// All System Equipment
// Adjust GVL_EquipArrays.cEQUIP_COUNT_MAX to accommodate all of the equipment to monitor
IF GVL_EquipArrays.nSystemEquip_Count <> 0 THEN
	FOR nStatusArrayIndex := 1 TO GVL_EquipArrays.nSystemEquip_Count BY 1 DO
		IF nStatusArrayIndex <= GVL_EquipArrays.cEQUIP_COUNT_MAX THEN
			// Only process the equipment if is is not in an offline state, this allows for the separate PLC equipment to 
			IF GVL_EquipArrays.aSystemEquipStatusArray[nStatusArrayIndex].CrntState <> E_StateCntrl.stOffline THEN
				// Test for an active warning on a coveyor
				IF GVL_EquipArrays.aSystemEquipStatusArray[nStatusArrayIndex].StsHasWarnings THEN
					ConveyorHasWarn := 1;
				END_IF
				// Test for an active Equipment fault, more than just a conveyor fault, could include Remote/IO, Barcode reader, etc..
				IF GVL_EquipArrays.aSystemEquipStatusArray[nStatusArrayIndex].StsFaulted THEN
					ConveyorHasFault := 1;
				END_IF
				// Test for a sleeping state
				IF GVL_EquipArrays.aSystemEquipStatusArray[nStatusArrayIndex].CrntOperState = E_OperStateCntrl.sleeping THEN
					ConveyorIsSleeping := 1;
				END_IF
				// Test for the Auto state, again an equipment state test to include non-conveyor equipment
				IF GVL_EquipArrays.aSystemEquipStatusArray[nStatusArrayIndex].StsAuto THEN
					ConveyorInAuto := 1;
				END_IF
			END_IF
		END_IF
	END_FOR
END_IF

// Initialise the Stack Light, only changing values as required
//GVL_IO.LT_MainPanelStack_Blue := FALSE;
GVL_IO.LT_MainPanelStack_Green := FALSE;
GVL_IO.LT_MainPanelStack_Yellow := FALSE;
GVL_IO.LT_MainPanelStack_Red := FALSE;
GVL_IO.LT_10161_Red := FALSE;
GVL_IO.LT_3131_Red := FALSE;
GVL_IO.LT_8181_Red := FALSE;
GVL_IO.LT_10171_Yellow := FALSE;
GVL_IO.LT_3151_Yellow := FALSE;
GVL_IO.LT_8191_Yellow := FALSE;
GVL_IO.LT_10201_Green := FALSE;
GVL_IO.LT_3201_Green := FALSE;
GVL_IO.LT_8231_Green := FALSE;
	
IF ConveyorHasFault OR NOT SystemSafety.Safety_SystemEstopsOK THEN
	// Red light SOLID ON
	GVL_IO.LT_MainPanelStack_Red := TRUE;
	GVL_IO.LT_10161_Red := TRUE;
	GVL_IO.LT_3131_Red := TRUE;
	GVL_IO.LT_8181_Red := TRUE;
ELSE
	IF ConveyorHasWarn THEN
		// Orange Light SOLID ON
		GVL_IO.LT_MainPanelStack_Yellow := TRUE;
		GVL_IO.LT_10171_Yellow := TRUE;
		GVL_IO.LT_3151_Yellow := TRUE;
		GVL_IO.LT_8191_Yellow := TRUE;
	ELSE
		IF ConveyorInAuto THEN
			// Green Light SOLID ON
			GVL_IO.LT_MainPanelStack_Green := TRUE;
			GVL_IO.LT_10201_Green := TRUE;
			GVL_IO.LT_3201_Green := TRUE;
			GVL_IO.LT_8231_Green := TRUE;
		ELSE
			GVL_IO.LT_MainPanelStack_Green := SysShrtPulseTmr.Output;
			GVL_IO.LT_10201_Green :=  SysShrtPulseTmr.Output;
			GVL_IO.LT_3201_Green :=  SysShrtPulseTmr.Output;
			GVL_IO.LT_8231_Green :=  SysShrtPulseTmr.Output;
		END_IF
	END_IF
	IF GVL_IO.HornMainPanel THEN
		// Orange Light FLASHING ON
		GVL_IO.LT_MainPanelStack_Yellow := SysShrtPulseTmr.Output;
		GVL_IO.LT_10171_Yellow := SysShrtPulseTmr.Output;
		GVL_IO.LT_3151_Yellow := SysShrtPulseTmr.Output;
		GVL_IO.LT_8191_Yellow := SysShrtPulseTmr.Output;
	END_IF;
END_IF

END_PROGRAM

// ---- FunctionBlocks/Utils/FB_SystemCntrl.TcPOU
FUNCTION_BLOCK FB_SystemCntrl

(* System Interlock and Event Set up,
	Uses Interlocks.
	Doesn't use Start Conditions or the horn delay  
	Uses Events
	
	This exists to allow the Interlock/Event descriptions and setup to be managed through the HMI
	and be easily setup as system faults.
*)
VAR_IN_OUT
	{attribute 'OPC.UA.DA' := '1'}
	Sts_EquipState				: ST_EquipmentStatus;		// State Status
END_VAR
VAR_INPUT
	{attribute 'OPC.UA.DA' := '1'}
	In_o_EquipStatePB			: ST_StateCntrlPB;		// Hmi push buttons to change states
	In_p_EquipStatePB			: ST_StateCntrlPB;		// Other push buttons to change states
	{attribute 'OPC.UA.DA' := '1'}
	Cfg_EquipLabel				: STRING(20);		// Label of the equipment
	// Events
	In_SystemEvents				: UINT;		// Event that is specific to the instance of the solenoid/actuator
	{attribute 'OPC.UA.DA' := '0'}
	Cfg_EquipEvntsArry			: ARRAY [0..15] OF ST_CfgEvents;
	
	// Interlocks that can be Instance Specific
	In_SystemIntlks				: UINT;		// Interlock that is specific to the instance of the solenoid/actuator
	{attribute 'OPC.UA.DA' := '0'}
	Cfg_EquipIntlksArry		: ARRAY [0..15] OF ST_CfgEvents;		// Descriptions of the Interlock 
	
END_VAR
VAR_OUTPUT
	{attribute 'OPC.UA.DA' := '1'}
	Out_Auto					:	BOOL;	// Combine HMI and Other Start/Auto signals to issue a single START/AUTO command
	{attribute 'OPC.UA.DA' := '1'}
	Out_Stop					:	BOOL;	// Combine HMI and Other Stop signals to issue a single STOP command
	{attribute 'OPC.UA.DA' := '1'}
	Out_Reset					:	BOOL;	// Combine HMI and Other Reset signals to issue a single RESET command
	{attribute 'OPC.UA.DA' := '1'}
	Sts_All_Intlks_OK			: BOOL;		// Status bit to show that all interloks are good to Run 
	{attribute 'OPC.UA.DA' := '1'}
	Sts_FaultActive				: BOOL;	// Status Bit Showing that a fault is present (0= No Active Faults, 1= Fault Active)
	{attribute 'OPC.UA.DA' := '1'}
	Sts_WarnActive				: BOOL;	// Status Bit Showing that a warning is present (0= No Active Warnings, 1= Warning Active)
	{attribute 'OPC.UA.DA' := '1'}
	Sts_All_Evnts_OK			: BOOL;		// Status Bit Showing that ALL Events are OK to RUN (0= Event Present, 1= OK to Run)
	{attribute 'OPC.UA.DA' := '1'}
	Sts_IntlksArry				: ARRAY[0..15] OF ST_EventSts;		// Interlock status 0 to 15 Input
	{attribute 'OPC.UA.DA' := '1'}
	Sts_FaultsArry				: ARRAY[0..15] OF ST_EventSts;	// Status of each Fault Event State (0= OFF, 1=ON)
	{attribute 'OPC.UA.DA' := '1'}
	Sts_WarnsArry				: ARRAY[0..15] OF ST_EventSts;		// Status of each Warning Event State (0= OFF, 1=ON)
	{attribute 'OPC.UA.DA' := '0'}
	Sts_EvntsArry				: ARRAY[0..15] OF ST_EventSts; 	// Status of each Event State (0= OFF, 1=ON)
END_VAR
VAR
	{attribute 'OPC.UA.DA' := '0'}
	System_fbIntrlks				: FB_Intlks_Latch;
	System_IntlksArry				: ARRAY[0..15] OF BOOL;
	{attribute 'OPC.UA.DA' := '0'}
	System_EventManager				: FB_EventMngr;
	System_EventArry				: ARRAY[0..15] OF BOOL;
	System_LatchIgnore				: BOOL := FALSE;		// Put as a place holder for ease of future use
	System_LatchReset				: BOOL := FALSE;		//Put as a place holder for ease of future use
	System_IntlkBypassed			: ARRAY [0..15] OF BOOL;		//Put as a place holder for ease of future use
END_VAR

// Set Up inputs for interlocks that are specific for the configuration instance
System_IntlksArry[0] := In_SystemIntlks.0;
System_IntlksArry[1] := In_SystemIntlks.1; 
System_IntlksArry[2] := In_SystemIntlks.2;
System_IntlksArry[3] := In_SystemIntlks.3;
System_IntlksArry[4] := In_SystemIntlks.4;
System_IntlksArry[5] := In_SystemIntlks.5;
System_IntlksArry[6] := In_SystemIntlks.6;
System_IntlksArry[7] := In_SystemIntlks.7;
System_IntlksArry[8] := In_SystemIntlks.8;
System_IntlksArry[9] := In_SystemIntlks.9; 
System_IntlksArry[10] := In_SystemIntlks.10;
System_IntlksArry[11] := In_SystemIntlks.11;
System_IntlksArry[12] := In_SystemIntlks.12;
System_IntlksArry[13] := In_SystemIntlks.13;
System_IntlksArry[14] := In_SystemIntlks.14;
System_IntlksArry[15] := In_SystemIntlks.15;
	
// Call Interlock block
System_fbIntrlks(
	In_Intlks:= System_IntlksArry,
	CFG_IntlksArry:= Cfg_EquipIntlksArry, 
	HMI_LatchIgnore:= System_LatchIgnore, 
	HMI_LatchReset:= System_LatchReset, 
	All_Intlk_OK=> Sts_All_Intlks_OK, 
	STS_Intlks=> Sts_IntlksArry);
	
System_EventArry[0]:= In_SystemEvents.0;
System_EventArry[1]:= In_SystemEvents.1;
System_EventArry[2]:= In_SystemEvents.2;
System_EventArry[3]:= In_SystemEvents.3;
System_EventArry[4]:= In_SystemEvents.4;
System_EventArry[5]:= In_SystemEvents.5;
System_EventArry[6]:= In_SystemEvents.6;
System_EventArry[7]:= In_SystemEvents.7;
System_EventArry[8]:= In_SystemEvents.8;
System_EventArry[9]:= In_SystemEvents.9;
System_EventArry[10]:= In_SystemEvents.10;
System_EventArry[11]:= In_SystemEvents.11;
System_EventArry[12]:= In_SystemEvents.12;
System_EventArry[13]:= In_SystemEvents.13;
System_EventArry[14]:= In_SystemEvents.14;
System_EventArry[15]:= In_SystemEvents.15;

// Event Manager
System_EventManager(
	sEquipStateCntrlSts := Sts_EquipState.Sts_EquipmentState,
	In_EventsArry := System_EventArry ,  
	CFG_EvntsArry:= Cfg_EquipEvntsArry, 
	HMI_LatchReset:= In_o_EquipStatePB.ResetPB OR In_p_EquipStatePB.ResetPB,
	Out_FaultActive=> Sts_FaultActive, 
	Out_WarnActive=> Sts_WarnActive, 
	Sts_All_Evnts_OK=> Sts_All_Evnts_OK, 
	Sts_FaultsArry=> Sts_FaultsArry, 
	Sts_WarnsArry=> Sts_WarnsArry, 
	Sts_EvntsArry=> Sts_EvntsArry);

// Activate the Out_ variables
Out_Auto := In_o_EquipStatePB.AutoPB OR In_p_EquipStatePB.AutoPB;
Out_Stop := In_o_EquipStatePB.StopPB OR In_p_EquipStatePB.StopPB;
Out_Reset := In_o_EquipStatePB.ResetPB OR In_p_EquipStatePB.ResetPB;

// Populate the Sts Output Variables
Sts_EquipState.Sts_EquipmentState.CrntState := 1;
Sts_EquipState.Sts_All_Intlks_OK  := Sts_All_Intlks_OK;
Sts_EquipState.Sts_All_Evnts_OK  := Sts_All_Evnts_OK;
Sts_EquipState.Sts_FaultActive := Sts_FaultActive;
Sts_EquipState.Sts_WarnActive := Sts_WarnActive;

END_FUNCTION_BLOCK

// ---- FunctionBlocks/Utils/Events/FB_Intlks_Latch.TcPOU
FUNCTION_BLOCK FB_Intlks_Latch
(*
=====================================================================
	Copyright ©  Syscon Automation.  All Rights Reserved.
	Version 1 Release 1 2018
=====================================================================
 
	This FB monitors 16 interlock inputs
	Each "Good or OK" State for each Interlock Input is configurable (Default is 0=OK, 1=trip)
	Interlocks may be configured to latch which require a Reset Command to clear (latching can be disabled)
	Interlocks may be configured as Bypassable.
 --------------------------------------------------------------------
*)
 
VAR_INPUT
	In_Intlks:	ARRAY[0..15] OF BOOL;		// Interlocks 0 to 15 Input
	CFG_IntlksArry:	ARRAY[0..15] OF ST_CfgEvents;		// Configuration of Interlocks
	HMI_LatchIgnore:	BOOL;		// Input to ignore all latching requirements
	HMI_LatchReset:	BOOL;		// Input to reset latching interlocks
END_VAR
VAR_OUTPUT
	All_Intlk_OK: BOOL;		// Status Bit Showing that ALL Interlocks are OK to RUN (either interlock is OK or it has been bypassed (0= Interlock Enabled-Stop, 1= OK to Run)	
	STS_Intlks:	ARRAY[0..15] OF ST_EventSts;		// Status of each Interlock State (0= OFF, 1=ON)
	STS_LatchResetReq:	BOOL;		// Status bit to show that latch reset is req
	STS_BypassActive: BOOL;		// Status Bit Showing that a Bypass is Active (0= No Active Bypass, 1= A Bypass is Active) 
	
END_VAR
VAR
	Intlk_CrntStsArry:	ARRAY[0..15] OF BOOL;		// The Current state of the interlock after compared to OK state
	Intlks_LatchedArry:	ARRAY[0..15] OF BOOL;		//Currently Latched ON
	Intlks_Bypassed:	ARRAY[0..15] OF BOOL;		// Interlocks where Bypass is ON and Allowed
	STS_LatchResetReqArry:	ARRAY[0..15] OF BOOL; 		// Status to see if latch reset is required (0= OFF, 1=ON)
	Sts_Intlks_BypassNotAllowed:	ARRAY[0..15] OF BOOL;		// Status representing each Non Bypassable Interlock State (0= OFF, 1=ON)
	IntlkRaw_ON:	BOOL;		// Testing Bit to Show that an Interlock is Active Based on Current OK State (ignoring Latches and Bypassing)
	Intlk_ON:	BOOL;		// Testing Bit to Show that an Interlock is Active Based on Current OK State (After Latches and Bypassing)
	i: INT;		//index
END_VAR

// Run loop to check each input
FOR i := 0 TO 15 DO
	// Compare to OK State
	Intlk_CrntStsArry[i] := In_Intlks[i] XOR CFG_IntlksArry[i].OKState;
	
	//Look at Latching
	IF HMI_LatchIgnore THEN
		Intlks_LatchedArry[i] := Intlk_CrntStsArry[i];
	ELSE
		Intlks_LatchedArry[i] := Intlk_CrntStsArry[i] OR CFG_IntlksArry[i].LatchRequired; 			
	END_IF
	
	//Set Status based on Latching
	STS_Intlks[i].Status := (STS_Intlks[i].Status AND Intlks_LatchedArry[i]) OR Intlk_CrntStsArry[i];
	STS_LatchResetReqArry[i] := (STS_Intlks[i].Status AND Intlks_LatchedArry[i] AND CFG_IntlksArry[i].LatchRequired);
	
	//Look for Bypass State
	Intlks_Bypassed[i] := CFG_IntlksArry[i].ByPssAllwd AND CFG_IntlksArry[i].HMI_BypassPB; 
	Sts_Intlks_BypassNotAllowed[i] := NOT Intlks_Bypassed[i];  
	Sts_Intlks_BypassNotAllowed[i] := Sts_Intlks_BypassNotAllowed[i] AND STS_Intlks[i].Status;
	
	//Update Status based on bypass
	STS_Intlks[i].Status := STS_Intlks[i].Status AND (NOT Intlks_Bypassed[i]);
	STS_Intlks[i].Description := CFG_IntlksArry[i].Description;
	STS_Intlks[i].DeviceLabel := CFG_IntlksArry[i].DeviceLabel;
	IF STS_Intlks[i].Status AND STS_Intlks[i].Description <> '' THEN
		STS_Intlks[i].StatusTxt := 'TRUE';
	ELSE
		STS_Intlks[i].StatusTxt := 'FALSE';
	END_IF
END_FOR

IF HMI_LatchReset THEN
	FOR i := 0 TO 15 DO
		STS_Intlks[i].Status := FALSE;
		STS_LatchResetReqArry[i] := FALSE;
	END_FOR
END_IF

//Set Up test bit showing all active interlocks ignoring
IntlkRaw_ON := In_Intlks[0] OR In_Intlks[1] OR In_Intlks[2] OR In_Intlks[3] 
			OR In_Intlks[4]OR In_Intlks[5] OR In_Intlks[6] OR In_Intlks[7]
			OR In_Intlks[8] OR In_Intlks[9] OR In_Intlks[10] OR In_Intlks[11]
			OR In_Intlks[12] OR In_Intlks[13] OR In_Intlks[14] OR In_Intlks[15];
			
// Set up bit showing that All interlocks are good			
Intlk_ON := STS_Intlks[0].Status OR STS_Intlks[1].Status OR STS_Intlks[2].Status OR STS_Intlks[3].Status
			OR STS_Intlks[4].Status OR STS_Intlks[5].Status OR STS_Intlks[6].Status OR STS_Intlks[7].Status
			OR STS_Intlks[8].Status OR STS_Intlks[9].Status OR STS_Intlks[10].Status OR STS_Intlks[11].Status
			OR STS_Intlks[12].Status OR STS_Intlks[13].Status OR STS_Intlks[14].Status OR STS_Intlks[15].Status;
	
//Set Up test bit showing that a latch is required
STS_LatchResetReq := NOT HMI_LatchIgnore AND (STS_LatchResetReqArry[0] OR STS_LatchResetReqArry[1] OR STS_LatchResetReqArry[2] OR STS_LatchResetReqArry[3] 
			OR STS_LatchResetReqArry[4]OR STS_LatchResetReqArry[5] OR STS_LatchResetReqArry[6] OR STS_LatchResetReqArry[7]
			OR STS_LatchResetReqArry[8] OR STS_LatchResetReqArry[9] OR STS_LatchResetReqArry[10] OR STS_LatchResetReqArry[11]
			OR STS_LatchResetReqArry[12] OR STS_LatchResetReqArry[13] OR STS_LatchResetReqArry[14] OR STS_LatchResetReqArry[15]);
						
// Set up bit showing that a bypass is active			
STS_BypassActive := Intlks_Bypassed[0] OR Intlks_Bypassed[1] OR Intlks_Bypassed[2] OR Intlks_Bypassed[3]
			OR Intlks_Bypassed[4] OR Intlks_Bypassed[5] OR Intlks_Bypassed[6] OR Intlks_Bypassed[7]
			OR Intlks_Bypassed[8] OR Intlks_Bypassed[9] OR Intlks_Bypassed[10] OR Intlks_Bypassed[11]
			OR Intlks_Bypassed[12] OR Intlks_Bypassed[13] OR Intlks_Bypassed[14] OR Intlks_Bypassed[15];
			
// Set up bit showing that All interlocks are good			
All_Intlk_OK := NOT( STS_Intlks[0].Status OR STS_Intlks[1].Status OR STS_Intlks[2].Status OR STS_Intlks[3].Status
			OR STS_Intlks[4].Status OR STS_Intlks[5].Status OR STS_Intlks[6].Status OR STS_Intlks[7].Status
			OR STS_Intlks[8].Status OR STS_Intlks[9].Status OR STS_Intlks[10].Status OR STS_Intlks[11].Status
			OR STS_Intlks[12].Status OR STS_Intlks[13].Status OR STS_Intlks[14].Status OR STS_Intlks[15].Status);

END_FUNCTION_BLOCK

// ---- FunctionBlocks/Utils/Events/FB_EventMngr.TcPOU
FUNCTION_BLOCK FB_EventMngr
(*
=====================================================================
	Copyright ©  Syscon Automation.  All Rights Reserved.
	Version 1 Release 2 2020
=====================================================================
 
	This FB monitors 16 Event inputs
	Each "Good or OK" State for each Event Input is configurable (Default is 0=OK, 1=trip)
	Events may be configured to latch which require a Reset Command to clear (latching can be disabled)
	Events may be configured as Warnings or Alarms)

	Release Notes: 2 - Added Equipment state/control/status reference and Stop codes to record Faults/Warnings to report to the System
						The Equipment reference was added because just adding the stop register as an array cannot compile (3.1.4022.32)
 --------------------------------------------------------------------
*)
VAR_IN_OUT
	sEquipStateCntrlSts: ST_StateCntrlSts;		// Equipment State, Control and Status Object
END_VAR 
VAR_INPUT
	In_EventsArry:	ARRAY[0..15] OF BOOL;		// Events 0 to 15 Input	
	CFG_EvntsArry:	ARRAY[0..15] OF ST_CfgEvents;		// Event Configuration 
	HMI_LatchIgnore:	BOOL;		// Input to ignore all latching requirements
	HMI_LatchReset:	BOOL;		// Input to reset latching Event
	
END_VAR
VAR_OUTPUT	
	Out_FaultActive:	BOOL;	// Status Bit Showing that a fault is present (0= No Active Faults, 1= Fault Active)
	Out_WarnActive:	BOOL;	// Status Bit Showing that a warning is present (0= No Active Warnings, 1= Warning Active)
	Sts_All_Evnts_OK: BOOL;		// Status Bit Showing that ALL Events are OK to RUN (0= Event Present, 1= OK to Run)
	Sts_FaultsArry:	ARRAY[0..15] OF ST_EventSts;		// Status of each Fault Event State (0= OFF, 1=ON)
	Sts_WarnsArry:	ARRAY[0..15] OF ST_EventSts;		// Status of each Warning Event State (0= OFF, 1=ON)
	Sts_EvntsArry:	ARRAY[0..15] OF ST_EventSts;		// Status of each Event State (0= OFF, 1=ON)
	Sts_LatchResetReq:	BOOL;		// Status bit to show that latch reset is req
	Sts_StopCode: UINT;				// Highest Priority Stop Code (Lowest Bit Weight)
	
END_VAR
VAR
	Evnt_CrntStsArry:	ARRAY[0..15] OF BOOL;		// The Current state of the Event after compared to OK state
	Evnts_LatchedArry:	ARRAY[0..15] OF BOOL;		//Currently Latched ON
	STS_LatchResetReqArry:	ARRAY[0..15] OF BOOL; 		// Status to see if latch reset is required (0= OFF, 1=ON)

	Evnt_ON:	BOOL;		// Testing Bit to Show that an Event is Active Based on Current OK State (ignoring Latches and Bypassing)
	i: INT;		//index
	fb_ManageStopCodes	:	FB_ManageCodes;			// Function Block with Methods to manage codes

	Evnt_Delay:		ARRAY[0..15] OF Tc2_Standard.TON;	// Set of timers to Delay configured events
	DelayTest:	DWORD;
END_VAR

// Clear the Sts_StopCode each pass
Sts_StopCode := 0;

// Run loop to check each input
FOR i := 0 TO 15 DO

	// Only "Online" items can be faulted
	IF sEquipStateCntrlSts.CrntState <> E_StateCntrl.stOffline THEN
		// Test for a value in the EventDelay
		DelayTest := TIME_TO_DWORD(CFG_EvntsArry[i].EventDelay); 
		IF ( DelayTest > 0) THEN
			Evnt_Delay[i].PT := CFG_EvntsArry[i].EventDelay;
			Evnt_Delay[i].IN := In_EventsArry[i] XOR CFG_EvntsArry[i].OKState;
			Evnt_Delay[i]();
			Evnt_CrntStsArry[i] := Evnt_Delay[i].Q;
		ELSE
			// Compare to OK State, if they match, the CrntStsArry is = 0
			//  1 XOR 1 = 0, 1 XOR 0 = 1, 0 XOR 1 = 1, 0 XOR 0 = 0 
			Evnt_CrntStsArry[i] := In_EventsArry[i] XOR CFG_EvntsArry[i].OKState;
		END_IF
	ELSE
		Evnt_CrntStsArry[i] := FALSE;
	END_IF
	
	//Look at Latching
	// HMI_LatchIgnore latches ALL Events, over-riding the Latch setup per event
	IF HMI_LatchIgnore THEN
		Evnts_LatchedArry[i] := Evnt_CrntStsArry[i];
	ELSE
		Evnts_LatchedArry[i] := Evnt_CrntStsArry[i] OR CFG_EvntsArry[i].LatchRequired; 			
	END_IF
	
	//Set Status based on Latching
	Sts_EvntsArry[i].Status := (Sts_EvntsArry[i].Status AND Evnts_LatchedArry[i]) OR Evnt_CrntStsArry[i];
	Sts_EvntsArry[i].Description := CFG_EvntsArry[i].Description;
	Sts_EvntsArry[i].DeviceLabel := CFG_EvntsArry[i].DeviceLabel;	
	STS_LatchResetReqArry[i] := (Sts_EvntsArry[i].Status AND Evnts_LatchedArry[i] AND CFG_EvntsArry[i].LatchRequired);
	IF Sts_EvntsArry[i].Status AND Sts_EvntsArry[i].Description <> '' THEN
		Sts_EvntsArry[i].StatusTxt := 'TRUE';
	ELSE
		Sts_EvntsArry[i].StatusTxt := 'FALSE';
	END_IF
	
	//Seperate into Alarms and Faults 
	Sts_FaultsArry[i].Status := Sts_EvntsArry[i].Status AND CFG_EvntsArry[i].FaultWarn;
	Sts_FaultsArry[i].Description := Sts_EvntsArry[i].Description;
	Sts_FaultsArry[i].DeviceLabel := Sts_EvntsArry[i].DeviceLabel;
	IF Sts_FaultsArry[i].Status AND Sts_FaultsArry[i].Description <> '' THEN
		Sts_FaultsArry[i].StatusTxt := 'TRUE';
	ELSE
		Sts_FaultsArry[i].StatusTxt := 'FALSE';
	END_IF
	
	Sts_WarnsArry[i].Status := Sts_EvntsArry[i].Status AND (NOT CFG_EvntsArry[i].FaultWarn);
	Sts_WarnsArry[i].Description := Sts_EvntsArry[i].Description;
	Sts_WarnsArry[i].DeviceLabel := Sts_EvntsArry[i].DeviceLabel;	
	IF Sts_WarnsArry[i].Status AND Sts_WarnsArry[i].Description <> '' THEN
		Sts_WarnsArry[i].StatusTxt := 'TRUE';
	ELSE
		Sts_WarnsArry[i].StatusTxt := 'FALSE';
	END_IF

	// Instanciate the fb_ManageStopCodes Function Block
	fb_ManageStopCodes(aCodeRegister := sEquipStateCntrlSts.stsStopRegister);

	// Check for a configured stop code
	IF CFG_EvntsArry[i].StopCode <> 0  THEN
		// Set the Stop Register for the configured stop code
		IF Sts_EvntsArry[i].Status THEN
			// Lowest Stop Code is highest Priority
			IF (Sts_StopCode > CFG_EvntsArry[i].StopCode) THEN
				Sts_StopCode := CFG_EvntsArry[i].StopCode;
			END_IF
			fb_ManageStopCodes.Set(nCodeToSet := CFG_EvntsArry[i].StopCode);
		ELSE
			// Clear the Stop Register for non-latching Events, when the HMI_LatchIgnore is NOT set
			IF NOT (CFG_EvntsArry[i].LatchRequired) AND NOT HMI_LatchIgnore THEN
				fb_ManageStopCodes.Clear(nCodeToClear := CFG_EvntsArry[i].StopCode);
			END_IF
		END_IF
	END_IF
	
END_FOR

IF HMI_LatchReset OR (sEquipStateCntrlSts.CrntState = E_StateCntrl.stOffline) THEN
	FOR i := 0 TO 15 DO
		Sts_EvntsArry[i].Status := FALSE;
		STS_LatchResetReqArry[i] := FALSE;
	END_FOR
	// When the Reset is issued, clear the entire stop register
	fb_ManageStopCodes.ClearRegister();
END_IF

//Set Up test bit showing all active Event ignoring bypasses and latching
Evnt_ON := In_EventsArry[0] OR In_EventsArry[1] OR In_EventsArry[2] OR In_EventsArry[3] 
			OR In_EventsArry[4]OR In_EventsArry[5] OR In_EventsArry[6] OR In_EventsArry[7]
			OR In_EventsArry[8] OR In_EventsArry[9] OR In_EventsArry[10] OR In_EventsArry[11]
			OR In_EventsArry[12] OR In_EventsArry[13] OR In_EventsArry[14] OR In_EventsArry[15];
			
//Set Up test bit showing that a latch is required
STS_LatchResetReq := NOT HMI_LatchIgnore AND (STS_LatchResetReqArry[0] OR STS_LatchResetReqArry[1] OR STS_LatchResetReqArry[2] OR STS_LatchResetReqArry[3] 
			OR STS_LatchResetReqArry[4]OR STS_LatchResetReqArry[5] OR STS_LatchResetReqArry[6] OR STS_LatchResetReqArry[7]
			OR STS_LatchResetReqArry[8] OR STS_LatchResetReqArry[9] OR STS_LatchResetReqArry[10] OR STS_LatchResetReqArry[11]
			OR STS_LatchResetReqArry[12] OR STS_LatchResetReqArry[13] OR STS_LatchResetReqArry[14] OR STS_LatchResetReqArry[15]);
						
// Set up bit showing that All Event are good			
STS_All_Evnts_OK := NOT( Sts_EvntsArry[0].Status OR Sts_EvntsArry[1].Status OR Sts_EvntsArry[2].Status OR Sts_EvntsArry[3].Status
			OR Sts_EvntsArry[4].Status OR Sts_EvntsArry[5].Status OR Sts_EvntsArry[6].Status OR Sts_EvntsArry[7].Status
			OR Sts_EvntsArry[8].Status OR Sts_EvntsArry[9].Status OR Sts_EvntsArry[10].Status OR Sts_EvntsArry[11].Status
			OR Sts_EvntsArry[12].Status OR Sts_EvntsArry[13].Status OR Sts_EvntsArry[14].Status OR Sts_EvntsArry[15].Status);

// Set up bit showing A Fault is Active			
Out_FaultActive := Sts_FaultsArry[0].Status OR Sts_FaultsArry[1].Status OR Sts_FaultsArry[2].Status OR Sts_FaultsArry[3].Status
			OR Sts_FaultsArry[4].Status OR Sts_FaultsArry[5].Status OR Sts_FaultsArry[6].Status OR Sts_FaultsArry[7].Status
			OR Sts_FaultsArry[8].Status OR Sts_FaultsArry[9].Status OR Sts_FaultsArry[10].Status OR Sts_FaultsArry[11].Status
			OR Sts_FaultsArry[12].Status OR Sts_FaultsArry[13].Status OR Sts_FaultsArry[14].Status OR Sts_FaultsArry[15].Status;
			
// Set up bit showing A Warning is Active			
Out_WarnActive :=  Sts_WarnsArry[0].Status OR Sts_WarnsArry[1].Status OR Sts_WarnsArry[2].Status OR Sts_WarnsArry[3].Status
			OR Sts_WarnsArry[4].Status OR Sts_WarnsArry[5].Status OR Sts_WarnsArry[6].Status OR Sts_WarnsArry[7].Status
			OR Sts_WarnsArry[8].Status OR Sts_WarnsArry[9].Status OR Sts_WarnsArry[10].Status OR Sts_WarnsArry[11].Status
			OR Sts_WarnsArry[12].Status OR Sts_WarnsArry[13].Status OR Sts_WarnsArry[14].Status OR Sts_WarnsArry[15].Status;

END_FUNCTION_BLOCK

// ---- FunctionBlocks/StateControl/FB_ManageCodes.TcPOU
FUNCTION_BLOCK FB_ManageCodes
VAR_IN_OUT
	aCodeRegister: ARRAY[*] OF UDINT;	// Variable array for Different sizes of Code Registers
END_VAR
VAR_INPUT
END_VAR
VAR_OUTPUT
END_VAR
VAR
	nBitIndex : UINT;						// Bit within the Word
	nArrayIndex : UINT;						// Word within the array
	nArrayTempIndex : UINT;					// Array Index for processing array
	nArrayCount : UINT;						// Number of words in the Array
	nUpdateValue : UDINT;					// Value of the Word to OR/XOR with the 
	nCheckValue : UDINT;					// Value of the Word to check with
	nBitCheck : UDINT;						// Word to use to check if a bit is set
	nLowerBitCheck : UDINT;					// Word to use to check if a lower weighted bit is set
END_VAR

VAR CONSTANT
	nBITCOUNT: UINT := 32;	// Number of Bits in each Array Element
	nBYTECOUNT : UINT := 4;	// Number of Bytes in each array element
END_VAR

// Get the array count
nArrayCount := (TO_UINT(SIZEOF(aCodeRegister)))/nBYTECOUNT;

METHOD PUBLIC Check : BOOL
VAR_INPUT
	nCodeToCheck : UINT;				// Code to Check For
END_VAR
VAR_OUTPUT
	bCodeSet : BOOL;					// Indicates that the Code is Set
	bHigherPriorityCode : BOOL;			// Indicates that a Higher Priority Code is Set
END_VAR
// Disable the warning regarding invalid Reference from a method for IO_OUT variables
{warning disable C0371}
// Test for a Valid reference
//IF __ISVALIDREF(aCodeRegister) THEN
	// Test to see if a bit is set
	nArrayIndex := 0;
	nBitIndex := 0;
	// Test for a valid value to test, > 0, < maximum number of available bits
	IF (nCodeToCheck <> 0) THEN
		IF nCodeToCheck <= (nArrayCount * nBITCOUNT) THEN
			// Use integer division to obtain the array index
			// Subtract 1 to put items in the range of 0-31 bits to use EXPT function to set individual bits (2^bit weight)
			nArrayIndex := (nCodeToCheck - 1) / nBITCOUNT;
			// Use modulo division to get the remainder that indicates the bit weight 
			nBitIndex := (nCodeToCheck - 1) MOD nBITCOUNT;
			// Calculate the value (2^nBitIndex)
			nCheckValue := TO_UDINT(EXPT(2,nBitIndex));
			// Bitwise AND the result with the target.
			// The AND clears all other bits in the word
			nBitCheck := aCodeRegister[nArrayIndex] AND nCheckValue;
			// The only bit that should survive the AND is the one we are checking for
			bCodeSet := (nBitCheck <> 0); 
		END_IF
	ELSE
		// Clear the Stop Code check when there is no request
		bCodeSet := 0;
	END_IF
	
	// Only test for a higher priority stop code if the tested stop code exists
	IF bCodeSet = 1 THEN
		// Test to see if a lower weighted bit is set
		nArrayIndex := 0;
		nBitIndex := 0;
		// Test for a valid value to test, > 0, < maximum number of available bits
		IF (nCodeToCheck <> 0) THEN
			IF nCodeToCheck <= (nArrayCount * nBITCOUNT) THEN
				// Use integer division to obtain the array index
				// Subtract 1 to put items in the range of 0-31 bits to use EXPT function to set individual bits (2^bit weight)
				nArrayIndex := (nCodeToCheck - 1) / nBITCOUNT;
				// Use modulo division to get the remainder that indicates the bit weight 
				nBitIndex := (nCodeToCheck - 1) MOD nBITCOUNT;
				// Calculate the value (2^nBitIndex)
				nCheckValue := TO_UDINT(EXPT(2,nBitIndex));
				// Subtract 1 from the bit we are checking, this flips all the less significant bits
				// E.g. 4 (0100b) - 1 (0001b) = 3 (0011b)
				// E.g. 21 (10101b) - 1 (00001b) = 20 (10100b)
				// E.g. 24 (11000b) - 1 (00001b) = 23 (10111b)
				nCheckValue := nCheckValue - 1; 
				// The AND masks out all bits above the specified weight, including the one we are testing for
				//  leaving only bits with a lower bit weight
				nLowerBitCheck := aCodeRegister[nArrayIndex] AND nCheckValue;
				// Test the calculated value for a lower bit
				bHigherPriorityCode := (nLowerBitCheck <> 0); 
				// Test to see if we are in the lowest array
				nArrayTempIndex := 0;
				IF nArrayIndex <> 0 THEN
					WHILE nArrayTempIndex < nArrayIndex  DO
						IF aCodeRegister[nArrayTempIndex] <> 0 THEN
							bHigherPriorityCode := 1;
						END_IF
						nArrayTempIndex := nArrayTempIndex + 1;
					END_WHILE
				END_IF
			END_IF
		END_IF
	ELSE
		// Reset the higher priority detected if the Tested Stop Code is not set
		bHigherPriorityCode := 0;
	END_IF
//END_IF
// Restore the warning regarding invalid Reference from a method for IO_OUT variables
{warning restore C0371}
END_METHOD

METHOD PUBLIC Clear
VAR_INPUT
	nCodeToClear : UINT;					// Stop Code to Activate
END_VAR
// Disable the warning regarding invalid Reference from a method for IO_OUT variables
{warning disable C0371}
// Test for a Valid reference
//IF __ISVALIDREF(aCodeRegister) THEN
	// Clear an individual bit
	// Initialize the index values
	nArrayIndex := 0;
	nBitIndex := 0;
	// Test for a valid value to test, > 0, < maximum number of available bits
	IF (nCodeToClear <> 0) THEN
		IF nCodeToClear <= (nArrayCount * nBITCOUNT) THEN
			// Use integer division to obtain the array index
			// Subtract 1 to put items in the range of 0-31 bits to use EXPT function to set individual bits (2^bit weight)
			nArrayIndex := (nCodeToClear - 1) / nBITCOUNT;
			// Use modulo division to get the remainder that indicates the bit weight 
			nBitIndex := (nCodeToClear - 1) MOD nBITCOUNT;
			// Calculate the value (2^nStopCode)
			nUpdateValue := TO_UDINT(EXPT(2,nBitIndex));
			// Bitwise OR the result with the target.
			// The OR leaves all other bits in the word set, even the one to be set if it already is
			// In this instance, it ensures that the following XOR clears the bit
			// 0 XOR 0 = 0, 1 XOR 0 = 0, 1 XOR 1 = 0
			aCodeRegister[nArrayIndex] := aCodeRegister[nArrayIndex] OR nUpdateValue;
			aCodeRegister[nArrayIndex] := aCodeRegister[nArrayIndex] XOR nUpdateValue; 
		END_IF
	END_IF
//END_IF
// Restore the warning regarding invalid Reference from a method for IO_OUT variables
{warning restore C0371}
END_METHOD

METHOD PUBLIC ClearRegister
VAR_INPUT
END_VAR
// Disable the warning regarding invalid Reference from a method for IO_OUT variables
{warning disable C0371}
// Test for a Valid reference
//IF __ISVALIDREF(aCodeRegister) THEN
	// aCodeRegister is a Zero based array
	// The SIZEOF will return the 1 based number of elements
	// Decrement this by 1 (one) to process the array
	FOR nArrayIndex := 0 TO (nArrayCount - 1) BY 1 DO
		// Clear each register
		aCodeRegister[nArrayIndex] := 0;
	END_FOR
//END_IF
// Restore the warning regarding invalid Reference from a method for IO_OUT variables
{warning restore C0371}
END_METHOD

METHOD PUBLIC Set
VAR_INPUT
	nCodeToSet	:	UINT;
END_VAR
// Disable the warning regarding invalid Reference from a method for IO_OUT variables
{warning disable C0371}
// Test for a Valid reference
//IF __ISVALIDREF(aCodeRegister) THEN
	// Set an individual bit
	// Initialize the index values
	nArrayIndex := 0;
	nBitIndex := 0;
	// Test for a valid value to test, > 0, < maximum number of available bits
	IF (nCodeToSet <> 0) THEN
		IF nCodeToSet <= (nArrayCount * nBITCOUNT) THEN
			// Use integer division to obtain the array index
			// Subtract 1 to put items in the range of 0-31 bits to use EXPT function to set individual bits (2^bit weight)
			nArrayIndex := (nCodeToSet - 1) / nBITCOUNT;
			// Use modulo division to get the remainder that indicates the bit weight 
			nBitIndex := (nCodeToSet - 1) MOD nBITCOUNT;
			// Calculate the value (2^nStopCode)
			nUpdateValue := TO_UDINT(EXPT(2,nBitIndex));
			// Bitwise OR the result with the target.
			// The OR leaves all other bits in the word set, even the one to be set if it already is
			aCodeRegister[nArrayIndex] := aCodeRegister[nArrayIndex] OR nUpdateValue;
		END_IF
	END_IF
//END_IF
// Restore the warning regarding invalid Reference from a method for IO_OUT variables
{warning restore C0371}
END_METHOD

END_FUNCTION_BLOCK

// ---- FunctionBlocks/Utils/FB_Flasher.TcPOU
(*
Function Block to vreate a flashing output.
If In_Trig goes TRUE the output will begin to blink On and OFF until In_Trig goes FALSE.
On duration is set by Cfg_OnTime
Off duration is set by Cfg_OffTime
*)
FUNCTION_BLOCK FB_Flasher
VAR_INPUT
	In_Trig:	BOOL;		// Input Trigger (1= Flsh output based on configured time intrevals)
	Cfg_OnTime:	TIME;		// Output On Time
	Cfg_OffTime:	TIME;	// Output Off Time
END_VAR
VAR_OUTPUT
	Output:	BOOL;		// Flashing Output
END_VAR
VAR
	StartTrig: R_TRIG;		// Rising Trigger
	OnTmrActive: BOOL;		// ON Timer active
	OnTmr: TON;				// ON Timer
	OffTmrActive: BOOL;		// OFF Timer active
	OffTmr: TON;			// OFF Timer
	StopTrig: F_TRIG;		// Falling Trigger 
END_VAR

// Start on Rise
StartTrig(CLK:= In_Trig);

IF StartTrig.Q THEN
	OnTmrActive := TRUE;
END_IF

// On timer
OnTmr(IN:= OnTmrActive, PT:= Cfg_OnTime);
IF OnTmr.Q THEN
	OnTmrActive := FALSE;
	OffTmrActive := TRUE;
END_IF

// Off Timer 
OffTmr(IN:= OffTmrActive, PT:= Cfg_OffTime);
IF OffTmr.Q THEN
	OnTmrActive := TRUE;
	OffTmrActive := FALSE;
END_IF

// Stop Trigger
StopTrig(CLK:= In_Trig);

IF StopTrig.Q THEN
	OnTmrActive := FALSE;
	OffTmrActive := FALSE;
END_IF

// Set Output
Output := OnTmrActive AND In_Trig;

END_FUNCTION_BLOCK

// ---- FunctionBlocks/Utils/FB_AlrtStrtDelay.TcPOU
(*
Function block to sound an Alert or Horn while delaying the start up of a piece of equipment
Can be controlled by a start and stop pulse In_StrtPulse/In_StpPulse Or by a holding the run variable In_Run TRUE.
The delay times are configured by CFG_AlertTime and CFG_WaitTime
The delay can be bypassed by In_BypssDelay.
If the run signal is True or the Start Pulse is triggered the Alert is sounded for the Alert time.
After Alert time is elapsed the alert is set to False and the wait time is then started
at the completion of the wait time the output is set to TRUE and the Out_Pulse is held true for one scan
If the In_BypssDelay input is true then the output is set to true imediately with the run signal or start pulse.
The alert can be fired manually (without affecting the delays) at anytime using the In_ManTstTrig input.
*)
FUNCTION_BLOCK FB_AlrtStrtDelay
VAR_INPUT
	In_Run:	BOOL;				// Run signal that has to be held on to operate delay
	In_StrtPulse :	BOOL;		// Pulse or Triger to Start Delay
	In_StpPulse :	BOOL;		// Pulse or Triger to Stop Delay
	CFG_AlertTime:	TIME;		// Time (or duration) for the alert or Horn to sound
	CFG_WaitTime:	TIME;		// Time to delay after alert or horn has sounded
	CFG_PulseTime:	TIME;		// Time to pulse the output signal
	In_ManTstTrig:	BOOL;		// Manual bit to alert or sound horn for the time/duration 
	In_BypssDelay:	BOOL;		// Input to disable and bypass alert or horn delay
END_VAR
VAR_OUTPUT
	Out:	BOOL;		// Output that is delayed by the horn timers.  Latched On while Run is True Or if RUN is FALSE then until Stop Pulse.
	Out_Pulse:	BOOL;		// Output that is delayed by the horn timers.  Pulsed for one scan
	Out_Timed:	BOOL;		// Output that is delayed by the horn timers.  Pulsed for configurable amount of time
	Out_Alert:	BOOL;		// Output for the ALert or Horn
	Sts_DelayActive:	BOOL; // Status output to show when output is actively being delayed
END_VAR
VAR
	AlertRequired: BOOL := FALSE;
	WaitRequired: BOOL := FALSE;
	AlertTon: TON;
	WaitActive: BOOL := FALSE;
	WaitTon: TON;
	DelayCompleted: BOOL := FALSE;
	DelayComplete: BOOL := FALSE;
	StartTrig: R_TRIG;
	ManTrig: R_TRIG;
	StopTrig: F_TRIG;
	OutTrig: R_TRIG;
	OutTrigTOF: TOF; // Pulse the Start Trigger for a set period of time
END_VAR

// Start Alert or Horn
StartTrig(CLK:= In_Run OR In_StrtPulse AND NOT In_BypssDelay);
IF StartTrig.Q THEN
	AlertRequired := TRUE;
	WaitRequired :=TRUE;
	Sts_DelayActive := TRUE;
END_IF

ManTrig(CLK:= In_ManTstTrig);
IF ManTrig.Q THEN
	AlertRequired := TRUE;
	WaitRequired :=FALSE;
END_IF

// Sound horn for timer
AlertTon(IN:= AlertRequired , PT:=CFG_AlertTime);

IF AlertTon.Q THEN
	AlertRequired:= FALSE;
	IF WaitRequired THEN
		WaitActive:= TRUE;
		DelayComplete := FALSE;	
	ELSE
		WaitActive := FALSE;
		WaitRequired := FALSE;
		Sts_DelayActive := FALSE;
		DelayComplete := TRUE;	
	END_IF	
END_IF

WaitTon(IN:=WaitActive, PT:=CFG_WaitTime);
IF WaitTon.Q THEN
	WaitActive := FALSE;
	WaitRequired := FALSE;
	Sts_DelayActive := FALSE;
	DelayComplete := TRUE;
END_IF

// Reset on stop
StopTrig(CLK:= In_Run OR In_StpPulse);
IF StopTrig.Q THEN
	AlertRequired:= FALSE;
	WaitRequired := FALSE;
	WaitActive := FALSE;
	Sts_DelayActive := FALSE;
	DelayComplete := FALSE;
END_IF
		
//Set Output
Out_Alert := AlertRequired;
Out := DelayComplete OR (In_BypssDelay AND In_Run);
OutTrig(CLK:= OUT, Q=> Out_Pulse);

// Timed Output
OutTrigTOF(IN := OutTrig.Q, PT := CFG_PulseTime);
Out_Timed := OutTrigTOF.Q;

END_FUNCTION_BLOCK

// ---- POUs/BarCodeReaders.TcPOU
PROGRAM BarCodeReaders
VAR
	BCR_S2140_01: CognexDataMan260;		// P2140 Divert 
	BCR_S2141_01: CognexDataMan260;		// P2141 Location Update
	BCR_S2150_01: CognexDataMan260;		// P2150 Sorter	
	BCR_S3080_01: CognexDataMan260;		// P3080 Location Update

//----------------------------------------BCR_S2140_01--------------------------------------------------------------		
	P2140_Arrival_Item 			: ST_Item;		// Output Item (Bar code read) To Sort PLC
	P2140_LastArrival_Item		: ST_Item;		// Last Output Item (Bar code read) To Sort PLC
	ReadID_P2140_Old		: UDINT;

	fb_SorterArrivalBuffer_P2140			: FB_ItemBuffer;	// Function to Process the SorterArrivalBuffer
	
	sBcr2140Log			: STRING;
	tpBcr2140Trig					: TP;	// Pulse timer for BCR Reader

	rSorter2140PE					: R_TRIG; 	// Capture the Rising edge of the Sorter BCR PE
	fSorter2140PE					: F_TRIG; 	// Capture the Falling edge of the Sorter BCR PE
	r_BCR2140TriggerON			: R_TRIG;
	f_BCR2140TriggerON			: F_TRIG;
	
//----------------------------------------BCR_S2150_01--------------------------------------------------------------
	P2150_Arrival_Item 			: ST_Item;		// Output Item (Bar code read) To Sort PLC
	P2150_LastArrival_Item		: ST_Item;		// Last Output Item (Bar code read) To Sort PLC
	ReadID_P2150_Old		: UDINT;

	fb_SorterArrivalBuffer_P2150			: FB_ItemBuffer;	// Function to Process the SorterArrivalBuffer

	sBcr2150Log			: STRING;
	tpBcr2150Trig					: TP;	// Pulse timer for BCR Reader

	rSorter2150PE					: R_TRIG; 	// Capture the Rising edge of the Sorter BCR PE
	fSorter2150PE					: F_TRIG; 	// Capture the Falling edge of the Sorter BCR PE
	r_BCR2150TriggerON			: R_TRIG;
	f_BCR2150TriggerON			: F_TRIG;

END_VAR

(*
	When multiple origination requests are possible, create multiple arrival buffers, one per origination request
	Along with all of the required structures 
	These additional buffers are mapped as I/O between this routine and the corresponding ProcessBuffers program instance
*)
//----------------------------------------BCR_S2140_01--------------------------------------------------------------
// Create instances of Buffer Processing Functions to initialize the buffers and data
fb_SorterArrivalBuffer_P2140.Master := TRUE;

// Setup Logging
fb_SorterArrivalBuffer_P2140.LogEntries := .nItemBufferLogEnable.ARRIVALS OR .nItemBufferLogEnableP2140.ARRIVALS;

// Setup Buffer Name for Logging
fb_SorterArrivalBuffer_P2140.Name := 'P2140 SYS ARRIVAL';

fb_SorterArrivalBuffer_P2140(st_BufferData := st_SorterArrivalBuffer_P2140
					, st_BufferFdbkIn := st_ArrivalFdbkIn_P2140
					, st_BufferFdbkOut => st_ArrivalFdbkOut_P2140);

IF GVL_IO.INIT THEN
	fb_SorterArrivalBuffer_P2140.Clear();
END_IF
//----------------------------------------BCR_S2150_01--------------------------------------------------------------
// Create instances of Buffer Processing Functions to initialize the buffers and data
fb_SorterArrivalBuffer_P2150.Master := TRUE;

// Setup Logging
fb_SorterArrivalBuffer_P2150.LogEntries := .nItemBufferLogEnable.ARRIVALS OR .nItemBufferLogEnableP2150.ARRIVALS;

// Setup Buffer Name for Logging
fb_SorterArrivalBuffer_P2150.Name := 'P2150 SYS ARRIVAL';

fb_SorterArrivalBuffer_P2150(st_BufferData := st_SorterArrivalBuffer_P2150
					, st_BufferFdbkIn := st_ArrivalFdbkIn_P2150
					, st_BufferFdbkOut => st_ArrivalFdbkOut_P2150);

IF GVL_IO.INIT THEN
	fb_SorterArrivalBuffer_P2150.Clear();
END_IF


// Reset All Metrics when requested
IF MAIN.In_ResetAllMetrics THEN
	BCR_S2140_01.In_ResetCounts := MAIN.In_ResetAllMetrics;
	BCR_S2141_01.In_ResetCounts := MAIN.In_ResetAllMetrics;
	BCR_S2150_01.In_ResetCounts := MAIN.In_ResetAllMetrics;
	BCR_S3080_01.In_ResetCounts := MAIN.In_ResetAllMetrics;

END_IF
//----------------------------------------BCR_S2140_01--------------------------------------------------------------
//Divert
// Set up Bar Code Readers
BCR_S2140_01.LogEntries := .nBarcodeLogEnable.BCR_S2140_01_LOG;
BCR_S2140_01(
	In_ReadTrig:= PhotoEyes.PE_10081.Out_OnFltrd, 
	In_ResetCounts:= , 
	In_TriggerOnTime := T#20MS ,
	In_EquipID := '00064',
	Out_NewReadTrig=> , 
	Out_ReadString=> , 
	Out_ReadStatus=> ,
	Out_ResultID=>, 
	MisreadCount=> , 
	GoodreadCount=> );
//Logging
BCR_S2140_01.LogEntries := .nBarcodeLogEnable.BCR_S2140_01_LOG;
tpBcr2140Trig(
	IN := PhotoEyes.PE_10081.Out,
				PT := T#10MS,
				Q =>);
// Capture rising and falling edge Triggers of the Sorter BCR Trigger PE
rSorter2140PE(CLK:= PhotoEyes.PE_10081.Out, Q =>);
fSorter2140PE(CLK:= PhotoEyes.PE_10081.Out, Q =>);

// Log the rising/falling edge of the Trigger
IF rSorter2140PE.Q OR fSorter2140PE.Q THEN
	IF nBarcodeLogEnable.TRIGGER_PE THEN
		// Write to the Error List
		ADSLOGSTR( msgCtrlMask := ADSLOG_MSGTYPE_HINT OR ADSLOG_MSGTYPE_LOG,
			msgFmtStr := 'Sort BCR PE Blocked : %s',
			strArg := BOOL_TO_STRING(PhotoEyes.PE_10081.Out)
			); 
	END_IF
END_IF

// Send Read Information to Sorter	
//	Creates Arrival message at sorter
IF ReadID_P2140_Old <> BarCodeReaders.BCR_S2140_01.GoodreadCount THEN
	P2140_Arrival_Item.UniqueID := BCR_S2140_01.Out_ResultID;
	P2140_Arrival_Item.ID := BCR_S2140_01.Out_ReadString;
	P2140_Arrival_Item.Status := E_StatusCode.UpdateRequested;
	P2140_Arrival_Item.DeviceID := BCR_S2140_01.In_EquipID;
	P2140_Arrival_Item.MessageType := E_MessageIds.Arrival_23;
	P2140_Arrival_Item.Destination := .P2140_DefaultDestination;
	P2140_Arrival_Item.Length := 0;
	P2140_LastArrival_Item := P2140_Arrival_Item;
	fb_SorterArrivalBuffer_P2140.AddItem(P2140_Arrival_Item);
	ReadID_P2140_Old := BarCodeReaders.BCR_S2140_01.GoodreadCount;
ELSE 
	P2140_Arrival_Item := BlankItem;
	P2140_Arrival_Item.Status := E_StatusCode.UpdateRequested;
END_IF

//----------------------------------------BCR_S2141_01--------------------------------------------------------------
//Location Update
// Set up Bar Code Readers
BCR_S2141_01.LogEntries := .nBarcodeLogEnable.BCR_S2141_01_LOG;
BCR_S2141_01(
	In_ReadTrig:= PhotoEyes.PE_10302.Out_OnFltrd, 
	In_ResetCounts:= , 
	In_TriggerOnTime := T#20MS ,
	In_EquipID := '00067',
	Out_NewReadTrig=> , 
	Out_ReadString=> , 
	Out_ReadStatus=> ,
	Out_ResultID=>, 
	MisreadCount=> , 
	GoodreadCount=> );
//----------------------------------------BCR_S2150_01--------------------------------------------------------------
//Sorter
// Set up Bar Code Readers
	BCR_S2150_01.LogEntries := .nBarcodeLogEnable.BCR_S2150_01_LOG;
	BCR_S2150_01(
	In_ReadTrig:= PhotoEyes.PE_2301.Out, 
	In_ResetCounts:= , 
	In_TriggerOnTime := T#20MS ,
	In_EquipID := '00081',
	Out_NewReadTrig=> , 
	Out_ReadString=> , 
	Out_ReadStatus=> ,
	Out_ResultID=>, 
	MisreadCount=> , 
	GoodreadCount=> );
//Logging	
BCR_S2150_01.LogEntries := .nBarcodeLogEnable.BCR_S2150_01_LOG;
tpBcr2150Trig(
	IN := PhotoEyes.PE_2301.Out,
				PT := T#10MS,
				Q =>);
// Capture rising and falling edge Triggers of the Sorter BCR Trigger PE
rSorter2150PE(CLK:= PhotoEyes.PE_2301.Out, Q =>);
fSorter2150PE(CLK:= PhotoEyes.PE_2301.Out, Q =>);

// Log the rising/falling edge of the Trigger
IF rSorter2150PE.Q OR fSorter2150PE.Q THEN
	IF nBarcodeLogEnable.TRIGGER_PE THEN
		// Write to the Error List
		ADSLOGSTR( msgCtrlMask := ADSLOG_MSGTYPE_HINT OR ADSLOG_MSGTYPE_LOG,
			msgFmtStr := 'Sort BCR PE Blocked : %s',
			strArg := BOOL_TO_STRING(PhotoEyes.PE_2301.Out)
			); 
	END_IF
END_IF

// Send Read Information to Sorter	
//	Creates Arrival message at sorter
IF ReadID_P2150_Old <> BarCodeReaders.BCR_S2150_01.GoodreadCount THEN
	P2150_Arrival_Item.UniqueID := BCR_S2150_01.Out_ResultID;
	P2150_Arrival_Item.ID := BCR_S2150_01.Out_ReadString;
	P2150_Arrival_Item.Status := E_StatusCode.UpdateRequested;
	P2150_Arrival_Item.DeviceID := BCR_S2150_01.In_EquipID;
	P2150_Arrival_Item.MessageType := E_MessageIds.Arrival_23;
	P2150_Arrival_Item.Destination := MsgControl.DefDestination;
	P2150_Arrival_Item.Length := 0;
	P2150_LastArrival_Item := P2150_Arrival_Item;
	fb_SorterArrivalBuffer_P2150.AddItem(P2150_Arrival_Item);
	ReadID_P2150_Old := BarCodeReaders.BCR_S2150_01.GoodreadCount;
ELSE 
	P2150_Arrival_Item := BlankItem;
	P2150_Arrival_Item.Status := E_StatusCode.UpdateRequested;
END_IF

//----------------------------------------BCR_S3080_01--------------------------------------------------------------
//Location Update
// Set up Bar Code Readers
BCR_S3080_01.LogEntries := .nBarcodeLogEnable.BCR_S3080_01_LOG;
	BCR_S3080_01(
	In_ReadTrig:= PhotoEyes.PE_9161.Out_OnFltrd, 
	In_ResetCounts:= , 
	In_TriggerOnTime := T#20MS ,
	In_EquipID := '00068',
	Out_NewReadTrig=> , 
	Out_ReadString=> , 
	Out_ReadStatus=> ,
	Out_ResultID=>, 
	MisreadCount=> , 
	GoodreadCount=> );

END_PROGRAM

// ---- FunctionBlocks/BarCode/CognexDataMan260.TcPOU
FUNCTION_BLOCK CognexDataMan260
VAR_INPUT
	{attribute 'OPC.UA.DA' := '1'}
	In_ResetMetrics		: BOOL;
	In_ReadTrig			: BOOL;			// Read Trigger input -- (1=Read Bar Code)
	In_ResetCounts		: BOOL;		// Trigger to reset counters (1=Reset)
	In_TriggerOnTime	: TIME := T#200MS;
	{attribute 'OPC.UA.DA' := '1'}
	In_EquipID			: STRING(20);	// Equip ID used for reporting
	
END_VAR
VAR_OUTPUT
	Out_NewReadTrig		: BOOL;		// Output trigger(single scan) to show a new read has just posted data to Out_ReadString (1=new read)
	{attribute 'OPC.UA.DA' := '1'}
	Out_ReadString		: STRING(30);	// String Output from Barcode read
	{attribute 'OPC.UA.DA' := '1'}
	Out_ReadStatus		: BOOL;		// Read Status stays latched if next read is the same (1=Good)
	{attribute 'OPC.UA.DA' := '1'}
	Out_ResultID		: INT;		// Read Count from Barcode Reader
	{attribute 'OPC.UA.DA' := '1'}
	Out_DeviceState		: UINT;		// Device Connection State 
	Out_TriggerState	: BOOL;
	{attribute 'OPC.UA.DA' := '1'}
	MisreadCount		: UDINT;		// Count for number of bad reads since startup
	{attribute 'OPC.UA.DA' := '1'}
	GoodreadCount		: UDINT;		// Count for number of good reads since startup
	{attribute 'OPC.UA.DA' := '1'}
	Out_LastTenReads	: ARRAY[1..10] OF STRING(30);	// Array of the last 10 barcodes decoded
	
END_VAR
VAR
	bLogEntries: BOOL := FALSE;		// If true, log entries
	ResultID_Old: INT;		// Variable used to detect change in read data
	DataReadCount: INT;		// Read Data Length Check length
	x: INT;		// index variable
	CharArry: ARRAY [0..DataBytesSize] OF STRING(2);		// Characters read in barcode
	DeviceState	AT %I* : UINT;	// Device Connection State -- From mapped DevState 
	TriggerReady	AT %I* : BOOL;	// Barcode Reader Mapped VAR
	TriggerAck	AT %I* : BOOL;	// Barcode Reader Mapped VAR
	Acquiring 	AT %I* : BOOL;	// Barcode Reader Mapped VAR
	Decoding 	AT %I* : BOOL;	// Barcode Reader Mapped VAR
	DecodeComplete 	AT %I* : BOOL;	// Barcode Reader Mapped VAR
	ResultsAvail	AT %I* : BOOL;	// Barcode Reader Mapped VAR
	TriggerID	AT %I*: INT;	// Barcode Reader Mapped VAR
	ResultID	AT %I* : INT;	// Barcode Reader Mapped VAR
	ResultCode	AT %I* : INT;	// Barcode Reader Mapped VAR
	ResultLength	AT %I* : INT;	// Barcode Reader Mapped VAR
	ResultData	AT %I* : ARRAY [0 .. DataBytesSize] OF BYTE;	// Barcode Reader Mapped VAR -- This ARRAY may be increased if more Data is needed 
	
	TriggerEnable	AT %Q*: BOOL;	// Barcode Reader Mapped VAR
	Trigger	AT %Q*: BOOL;	// Barcode Reader Mapped VAR
	ResultsAck	AT %Q*: BOOL;	// Barcode Reader Mapped VAR
	ResetTrigger: R_TRIG;
	TimeTestTrigger	: UINT;  // Variable used bitwise for all of the time testing triggers
	TriggerTime : TIME;
	TriggerAckTime: TIME;
	ResultsAvailTime: TIME;
	TotalTriggerTime: TIME;
	TotalResultsTime: TIME;
	ReadTrig_Trigger: R_TRIG;
	TriggerOnTimer: TON;
	TriggerPulse: TP;
	b_TempTrigger: BOOL;
END_VAR
VAR CONSTANT
	DataBytesSize	:INT := 25;
	GoodRead	:INT := 0;
	Validated	:INT := 1;
	Verified	:INT := 2;
	AcqTrigOverrun	:INT := 3;
	AcqBufferOverflow	:INT := 4;


END_VAR

(* Pass through Device state Left here in case future manipulation or more specific error codes are needed
	Bar Code Reader State Defined 
		0x8000 = Remote Node has no connections, 
		0x4000 = Remote Node is not reachable,
	 	0x2000 = TCP Client: initialization failed
		0x1000 = UDP Client: initialization failed
		0x0X00 = reserved
		0x0001 = 1st Connection disconnected
		0x0002 = 2nd Connection disconnected
		0x0004 = 3rd Connection disconnected
----------------------------------------------------*)
Out_DeviceState := DeviceState;

// Reset the metrics when Requested
IF In_ResetMetrics THEN
	MisReadCount := 0;
	GoodReadCount := 0;
	In_ResetMetrics := 0;
END_IF

// Set Reader to enable external trigger
TriggerEnable := TRUE;

// Watch Function Block for triggers
ResetTrigger(CLK:= In_ResetCounts);

// Reset single scan variable
IF Out_NewReadTrig THEN Out_NewReadTrig := FALSE; END_IF

//Set to only read on Rise
ReadTrig_Trigger(CLK:= In_ReadTrig);

// Fire Bar Code on read trigger
IF TriggerEnable AND TriggerReady AND ReadTrig_Trigger.Q THEN
	Trigger := TRUE;
	b_TempTrigger := TRUE;
	// Set Time capture for communications testing
	IF TimeTestTrigger.0 = FALSE THEN
		TriggerTime := TIME();
		TimeTestTrigger.0 := TRUE;
	END_IF

END_IF

// Reset the Temporary trigger
IF b_TempTrigger AND NOT In_ReadTrig THEN
	b_TempTrigger := FALSE;
END_IF
TriggerOnTimer(IN:= Trigger, PT:= IN_TriggerOnTime);
//TriggerOnTimer(IN:= b_TempTrigger, PT:= IN_TriggerOnTime);

TriggerPulse(IN := b_TempTrigger, PT := In_TriggerOnTime);

IF Trigger THEN
	IF TriggerOnTimer.Q  THEN
		Trigger := FALSE;
	END_IF
	
	// Set Time capture for communications testing
	IF TriggerAck AND TimeTestTrigger.1 = FALSE THEN
		TriggerAckTime := TIME();
		TimeTestTrigger.1 := TRUE;
	END_IF	
END_IF

//Trigger := TriggerPulse.Q;

Out_TriggerState := Trigger;

// Watch for Results
IF ResultsAvail AND ResultID_Old <> ResultID  THEN
	// Set Time capture for communications testing
	IF TimeTestTrigger.2 = FALSE THEN
		ResultsAvailTime := TIME();
		TimeTestTrigger.2 := TRUE;
	END_IF
	// Clear Old read
	Out_ReadString := '';
	// Make sure data from barcode fits in array 
	IF ResultLength > DataBytesSize THEN
		DataReadCount := DataBytesSize;
	ELSE 
		DataReadCount := ResultLength;
	END_IF
	
	// Set Read Status
	Out_ReadStatus := ResultCode.GoodRead;
	
	// Watch Counts
	IF ResultCode.GoodRead THEN
		GoodreadCount := GoodreadCount +1;
	ELSE
		MisreadCount := MisreadCount +1;
	END_IF
		
	FOR x := 0 TO DataReadCount DO
		CharArry[x] := F_ToCHR(ResultData[x]);
		Out_ReadString := CONCAT(STR1:= Out_ReadString , STR2:= CharArry[x] );
	END_FOR

	// Rotate the last read buffer
	FOR x := 9 TO 1 BY -1 DO
		Out_LastTenReads[x+1] := Out_LastTenReads[x];
	END_FOR

	Out_LastTenReads[1] := Out_ReadString;
	
	IF bLogEntries THEN
		logitem(Out_ReadString);
	END_IF	
	
	// Set trigger for new read
	Out_NewReadTrig := TRUE;
	// Reset Scan variables and BCR Acknowledge bit	
	Trigger := FALSE;
//	ResultsAck := FALSE;
	ResultsAck := TRUE; 			// Acknowledge that the results were read
	Out_ResultID := ResultID;		// Update the Output of the read count to show that a read was tried
	ResultID_Old := ResultID;

	// Calculate time results
	IF TimeTestTrigger.3 = FALSE THEN
		TotalTriggerTime := TriggerAckTime-TriggerTime;
		TotalResultsTime := ResultsAvailTime-TriggerTime;
		TimeTestTrigger.3 := TRUE;
	END_IF
 
END_IF

//Reset the Result Ack
IF NOT ResultsAvail THEN
	ResultsAck := FALSE;
END_IF

// Reset Counts
IF ResetTrigger.Q THEN
	GoodreadCount := 0;
	MisreadCount := 0;
END_IF

PROPERTY PUBLIC LogEntries : BOOL
GET
LogEntries := bLogEntries;
END_GET
SET
bLogEntries	 := LogEntries;
END_SET
END_PROPERTY

METHOD PRIVATE LogItem
VAR_INPUT
	s_Barcode			: STRING;
END_VAR

VAR
	sTempField			: STRING;
	sTempLogData		: STRING(255);
	nStatus				: INT;
	Out_ReadString		: INT;
END_VAR
sTempField := CONCAT(' Location: ', In_EquipID);
sTempField := CONCAT(sTempField,' Read: ');
sTempField := CONCAT(sTempField, s_Barcode);
// Write to the Error List
ADSLOGSTR( msgCtrlMask := ADSLOG_MSGTYPE_HINT OR ADSLOG_MSGTYPE_LOG
		, msgFmtStr := 'Barcode %s'
		, strArg := sTempField);
END_METHOD

END_FUNCTION_BLOCK

// ---- FunctionBlocks/Item/FB_ItemBuffer.TcPOU
FUNCTION_BLOCK FB_ItemBuffer
VAR_IN_OUT
	st_BufferData	:	ST_ItemBuffer;	// Buffer Type
END_VAR
VAR_INPUT
	st_BufferFdbkIn : ST_ItemBufferFdbk;	//	Buffer Feedback
END_VAR
VAR_OUTPUT
	// Output the In and Out pointer to allow testing of the 
	st_BufferFdbkOut : ST_ItemBufferFdbk;	//	Buffer Feedback
END_VAR
VAR
	nOutPointer		:	UDINT;				// OutPointer use to detect items in the buffer
	nBufferSizeTemp : 	UDINT;				// Calculate buffer size from Byte count
	nBufferSize : 	UDINT;					// Buffer Size in total elements
	st_Blank	:	ST_Item :=  (ID := '',
									UniqueID := 0,
									Destination := 0,
									Status := E_StatusCode.No_Status,
									DeviceID := '');
	nInit				: UDINT;					// Used to initialize the Array on Start-up
	nItemExtSize		: UDINT;				// Size of ST_ItemExt in Bytes
	bInitDone			: BOOL := FALSE;			// Set if Init occurred outside of FB_init
	bMaster				: BOOL := TRUE;			// Master = TRUE if this FB instance adds items to the buffer
	bLogEntries			: BOOL := FALSE;
	sBufferName			: STRING;				// Name of the Buffer for Logging Purposes
END_VAR

VAR CONSTANT
	nBITCOUNT: UINT := 32;	// Number of Bits in each Array Element
	nBYTECOUNT : UINT := 4;	// Number of Bytes in each array element
	nUDINTBYTECOUNT : UINT := 4;	// Number of Bytes in a UDINT data type
END_VAR

// This will run if FB_init did not detect a valid reference and initialize the Structure
IF NOT bInitDone THEN
(*
	// Get the Data Item In Bytes
	nBufferSizeTemp := TO_UDINT(SIZEOF(st_BufferData));
	// Reduce the byte count by the In and Out pointer byte count
	nBufferSizeTemp := nBufferSizeTemp - (nUDINTBYTECOUNT);
	// Get the size of the ST_ItemExt Data type
	nItemExtSize := TO_UDINT(SIZEOF(st_Blank));
	// Get the total number of bytes in the Array, by dividing the remaining nBufferSize by the nItemExtSize
	nBufferSize := nBufferSizeTemp/nItemExtSize;
*)
	nBufferSize := GetBufferSize();
	// Clear the buffer for the master
	// Set the OutPointer for a reader/consumer
	IF bMaster THEN
		// Clear the Buffer on Start-up because we don't know what is and is not in process
		clear();
	ELSE
		// If this is consumer, just start at the latest data point
		nOutPointer := st_BufferData.nInPointer;
	END_IF
(*
	FOR nInit := 0 TO (nBufferSize - 1) DO
		st_BufferData.aBufferData[nInit] := st_Blank;
	END_FOR 
	// Clear the Buffer In and Out pointers
	st_BufferData.nInPointer := 0;
	nOutPointer := 0;
	// Indicate that initialization occurred outside of FB_Init
	bInitDone := TRUE;
	// The master controls the buffer contents, when the buffer is clear, turn on the bClear bit
	IF bMaster THEN
		st_BufferData.bClear := TRUE;
	END_IF
	// Turn on the Buffer Empty signal regardless of Master status.
	// In system where there is no inter-plc communication, there will be no need for a non-master
	// function blocks 
	st_BufferFdbkOut.bEmpty := TRUE;
*)
	bInitDone := TRUE;
END_IF

// If this is the master and the feedback indicates that the consumer function blocks are empty
// clear the request
IF bMaster THEN
	IF st_BufferFdbkIn.bEmpty THEN
		st_BufferData.bClear := FALSE;
	END_IF
ELSE
	// If this is a consumer function block
	// Clear the buffer, even though this is all read from the master
	// the OutPointer is set to zero in the Clear method
	IF st_BufferData.bClear THEN
		Clear();
	ELSE
		st_BufferFdbkOut.bEmpty := FALSE;
	END_IF	
END_IF

METHOD PUBLIC AddItem : ST_Item
VAR_INPUT
	st_ItemToAdd	:	ST_Item;
END_VAR
// Disable the warning regarding invalid Reference from a method for IO_OUT variables
{warning disable C0371}
// Test for a Valid reference
IF __ISVALIDREF(st_BufferData) THEN
	// Increment the In Pointer using the F_CaclculateIndex
	st_BufferData.nInPointer := F_CalculateIndex(Offset := 1,InitialValue := st_BufferData.nInPointer, BufferSize := nBufferSize);
	// Add the Item to the Buffer
	st_BufferData.aBufferData[st_BufferData.nInPointer] := st_ItemToAdd;
	IF bLogEntries THEN
		logItem(bIn := TRUE
				, st_ItemToLog := st_ItemToAdd
				, nIndex := st_BufferData.nInPointer);
	END_IF
END_IF
// Restore the warning regarding invalid Reference from a method for IO_OUT variables
{warning restore C0371}
END_METHOD

PROPERTY PUBLIC BufferSize : UDINT
GET
BufferSize := nBufferSize;
END_GET
END_PROPERTY

METHOD PUBLIC Clear
VAR_INPUT
END_VAR
// Disable the warning regarding invalid Reference from a method for IO_OUT variables
{warning disable C0371}
// Test for a Valid reference
IF __ISVALIDREF(st_BufferData) THEN
	FOR nInit := 0 TO (nBufferSize - 1) DO
		st_BufferData.aBufferData[nInit] := st_Blank;
	END_FOR 
	// Clear the Buffer In and Out pointers
	st_BufferData.nInPointer := 0;
	nOutPointer := 0;
	// The master controls the buffer contents, when the buffer is clear, turn on the bClear bit
	IF bMaster THEN
		st_BufferData.bClear := TRUE;
	END_IF
	// Turn on the Buffer Empty signal regardless of Master status.
	// In system where there is no inter-plc communication, there will be no need for a non-master
	// function blocks 
	st_BufferFdbkOut.bEmpty := TRUE;
END_IF
// Restore the warning regarding invalid Reference from a method for IO_OUT variables
{warning restore C0371}
END_METHOD

METHOD FB_init : BOOL
VAR_INPUT
	bInitRetains : BOOL; // if TRUE, the retain variables are initialized (warm start / cold start)
	bInCopyCode : BOOL;  // if TRUE, the instance afterwards gets moved into the copy code (online change)
END_VAR
// ALWAYS ReInit the arrays
bInitDone := FALSE;
// Disable the warning regarding invalid Reference from a method for IO_OUT variables
{warning disable C0371}
// Test for a Valid reference
IF __ISVALIDREF(st_BufferData) THEN
(*
	// Get the Data Item In Bytes
	nBufferSizeTemp := TO_UDINT(SIZEOF(st_BufferData));
	// Reduce the byte count by the In and Out pointer byte count
	nBufferSizeTemp := nBufferSizeTemp - (nUDINTBYTECOUNT);
	// Get the size of the ST_ItemExt Data type
	nItemExtSize := TO_UDINT(SIZEOF(st_Blank));
	// Get the total number of bytes in the Array, by dividing the remaining nBufferSize by the nItemExtSize
	nBufferSize := nBufferSizeTemp/nItemExtSize;
*)
	nBufferSize := GetBufferSize();
	// Clear the Buffer on Start-up because we don't know what is and is not in process
	clear();
(*
	FOR nInit := 0 TO (nBufferSize - 1) DO
		st_BufferData.aBufferData[nInit] := st_Blank;
	END_FOR 
	// Clear the Buffer In and Out pointers
	st_BufferData.nInPointer := 0;
	nOutPointer := 0;
	// The master controls the buffer contents, when the buffer is clear, turn on the bClear bit
	IF bMaster THEN
		st_BufferData.bClear := TRUE;
	END_IF
	// Turn on the Buffer Empty signal regardless of Master status.
	// In system where there is no inter-plc communication, there will be no need for a non-master
	// function blocks 
	st_BufferFdbkOut.bEmpty := TRUE;
*)
END_IF

// Restore the warning regarding invalid Reference from a method for IO_OUT variables
{warning restore C0371}
END_METHOD

METHOD PRIVATE GetBufferSize : UDINT
VAR_INPUT
END_VAR
// Disable the warning regarding invalid Reference from a method for IO_OUT variables
{warning disable C0371}
// Test for a Valid reference
IF __ISVALIDREF(st_BufferData) THEN
	// Get the Data Item In Bytes
	nBufferSizeTemp := TO_UDINT(SIZEOF(st_BufferData));
	// Reduce the byte count by the In and Out pointer byte count
	nBufferSizeTemp := nBufferSizeTemp - (nUDINTBYTECOUNT);
	// Get the size of the ST_ItemExt Data type
	nItemExtSize := TO_UDINT(SIZEOF(st_Blank));
	// Get the total number of bytes in the Array, by dividing the remaining nBufferSize by the nItemExtSize
	nBufferSize := nBufferSizeTemp/nItemExtSize;
	GetBufferSize := nBufferSize;
END_IF

// Restore the warning regarding invalid Reference from a method for IO_OUT variables
{warning restore C0371}
END_METHOD

PROPERTY PUBLIC LogEntries : BOOL
GET
LogEntries := bLogEntries;
END_GET
SET
bLogEntries	 := LogEntries;
END_SET
END_PROPERTY

METHOD PRIVATE LogItem
VAR_INPUT
	bIn					: BOOL;
	st_ItemToLog		: ST_Item;
	nIndex				: UDINT;
END_VAR

VAR
	sTempField			: STRING;
	sTempLogData		: STRING(255);
	nStatus			: INT;
	Out_ReadString		: INT;
END_VAR
(*
	ID : STRING := '';		// Bar Code 	
	UniqueID : DINT := 0;		// Generic ID for tracking
	Destination : DINT := 0;
	Length : DINT := 0;
	Status : E_StatusCode := E_StatusCode.No_Status;
	CapturedInMetrics : BOOL;
	DeviceID:	STRING(5);	// Device ID associated with this record
	MessageType:	E_MessageIds;	// Message Type associated with this record
*)
// Prefix with the Direction 
IF bIn THEN
	sTempLogData := '>> ';
ELSE
	sTempLogData := '<< ';
END_IF

// Buffer Name
sTempField := CONCAT(sBufferName , ' ');
sTempLogData := CONCAT(sTempLogData, sTempField);

// Index
sTempField := CONCAT(UDINT_TO_STRING(nIndex), ' ');
sTempLogData := CONCAT(sTempLogData, sTempField);

// ID
sTempField := CONCAT(st_ItemToLog.ID, ' ');
sTempLogData := CONCAT(sTempLogData, sTempField);

// Unique ID
sTempField := CONCAT(DINT_TO_STRING(st_ItemToLog.UniqueID), ' ');
sTempLogData := CONCAT(sTempLogData, sTempField);

// Destination
sTempField := CONCAT(DINT_TO_STRING(st_ItemToLog.Destination), ' ');
sTempLogData := CONCAT(sTempLogData, sTempField);

// Status
nStatus := st_ItemToLog.Status;
sTempField := CONCAT(INT_TO_STRING(nStatus), ' ');
sTempLogData := CONCAT(sTempLogData, sTempField);

// DeviceID
sTempField := CONCAT(st_ItemToLog.DeviceID, ' ');
sTempLogData := CONCAT(sTempLogData, sTempField);

// MessageType
nStatus := st_ItemToLog.MessageType;
sTempLogData := CONCAT(sTempLogData, INT_TO_STRING(nStatus));

ADSLOGSTR( msgCtrlMask := ADSLOG_MSGTYPE_HINT OR ADSLOG_MSGTYPE_LOG
		, msgFmtStr := '%s'
		, strArg := sTempLogData);
END_METHOD

PROPERTY PUBLIC Master : BOOL
GET
Master := bMaster;
END_GET
SET
bMaster := Master;
END_SET
END_PROPERTY

PROPERTY PUBLIC Name : STRING
GET
Name := sBufferName;
END_GET
SET
sBufferName := Name;
END_SET
END_PROPERTY

PROPERTY PUBLIC OutPointer : UDINT
GET
OutPointer := nOutPointer;
END_GET
END_PROPERTY

METHOD PUBLIC RemoveItem : ST_Item
VAR_OUTPUT
	st_ItemToReturn	:	ST_Item;
END_VAR
// Disable the warning regarding invalid Reference from a method for IO_OUT variables
{warning disable C0371}
// Test for a Valid reference
IF __ISVALIDREF(st_BufferData) THEN
	// Allow items out of the buffer only when not being commanded to clear the buffer
	IF NOT st_BufferData.bClear THEN
		// Increment the In Pointer using the F_CaclculateIndex
		nOutPointer := F_CalculateIndex(Offset := 1,InitialValue := nOutPointer, BufferSize := nBufferSize);
		// Add the Item to the Buffer
		st_ItemToReturn := st_BufferData.aBufferData[nOutPointer];
		IF bLogEntries THEN
			logItem(bIn := FALSE
					, st_ItemToLog := st_ItemToReturn
					, nIndex := nOutPointer);
		END_IF
	END_IF
END_IF
// Restore the warning regarding invalid Reference from a method for IO_OUT variables
{warning restore C0371}
END_METHOD

END_FUNCTION_BLOCK

// ---- FunctionBlocks/Utils/F_CalculateIndex.TcPOU
(*
	This function calculates an index within an array using the max array size, 
	and the offset that you are looking for. This allows you to easily treat the array like a ring buffer
	For this function to work properly, the following rules MUST be observed
	1) The value in OFFSET will define the direction the index is adjusted
		> 0 Index is adjusted positively
		< 0 Index is adjusted negatively
	2)  InitialValue and BufferSize are both unsigned
	3) BufferSize is the number of elements in an array, not the maximum array index
		An array defined as ARRAY[0..10] has 11 elements, not 10, as the maximum element implies
		If the array is defined as [0..ARRAYMAX], where ARRAYMAX is a constant, BufferSize = ARRAYMAX + 1
*)
FUNCTION F_CalculateIndex : UDINT 
VAR_INPUT
	Offset			: DINT; //The offset that you want to calculate, the sign in important to indicate direction
	InitialValue	: UDINT; //The original point in the array you want to evaluate
	BufferSize		: UDINT; //The size of the array, not the index of the last array element
END_VAR
VAR
	TempInitialValue : LINT;
	TempIndex : LINT; //the calculation of the offset, before taking into account the size of the array, no wraparound
END_VAR

// Convert the InitialValue (UDINT) to a LINT to prevent sign changes due to implicit conversions
TempInitialValue := UDINT_TO_LINT(InitialValue); 
(*
	Calculate the new index, always add the Offset assuming the user correctly applied the sign
	 to indicate which direction to adjust the InitialValue
*)
TempIndex := TempInitialValue + Offset;

// Test the TempIndex to determine what the return index should be
// If it is zero or greater, test against the BufferSize value
IF TempIndex >= 0 THEN
	IF TempIndex >= BufferSize THEN 
		// If TempIndex is greater than the array size, reduce it by the BufferSize value
		F_CalculateIndex := LINT_TO_UDINT(TempIndex - BufferSize);
	ELSE
		// Return the TempIndex, it is with the bounds of the Array
		f_CalculateIndex := LINT_TO_UDINT(TempIndex);
	END_IF
ELSE
	// If the TempIndex value is negative, Add BufferSize to TempIndex and return the result
	F_CalculateIndex := LINT_TO_UDINT(BufferSize + TempIndex);
END_IF

END_FUNCTION

// ---- POUs/Photoeyes.TcPOU
PROGRAM Photoeyes
VAR
	DebounceOnTime:	TIME := T#500MS;     // Default Value
	DebounceOffTime:	TIME := T#500MS;     // Default Value
	JamDetectTime:	TIME := T#5S;     // Default Value
	
//----------------------------------------Photoeyes-----------------------------------------	
PE_2101   : FB_PhotoEye;  //P2150 FULL PHOTOEYE
PE_2131   : FB_PhotoEye;  //P2150 INDUCT PE SORTER PHOTOEYE
PE_2201   : FB_PhotoEye;  //P2146 FULL PHOTOEYE
PE_2231   : FB_PhotoEye;  //P2145 EXIT PHOTOEYE
PE_2301   : FB_PhotoEye;  //S2150 TRIGGER PHOTOEYE
PE_2331   : FB_PhotoEye;  //P2150 PE SINGULATION GRABBER TRIGGER PHOTOEYE
PE_3111   : FB_PhotoEye;  //P2150-02 TRANSFER COMPLETED PHOTOEYE
PE_3231   : FB_PhotoEye;  //P2150-01 TRANSFER COMPLETED PHOTOEYE
PE_4091   : FB_PhotoEye;  //P2150-04 TRANSFER COMPLETED PHOTOEYE
PE_4161   : FB_PhotoEye;  //P2150 SORTER DISCHARGE PHOTOEYE
PE_4201   : FB_PhotoEye;  //P2150-03 TRANSFER COMPLETED PHOTOEYE
PE_8131   : FB_PhotoEye;  //P2141 EXIT PHOTOEYE
PE_8141   : FB_PhotoEye;  //P2142 FULL PHOTOEYE
PE_8161   : FB_PhotoEye;  //P2143 EXIT PHOTOEYE
PE_9141   : FB_PhotoEye;  //P3080 EXIT PHOTOEYE
PE_9161   : FB_PhotoEye;  //S3080-01 TRIGGER PHOTOEYE
PE_9191   : FB_PhotoEye;  //P3080 EXIT PHOTOEYE
PE_9221   : FB_PhotoEye;  //P3080 HEIGHT CHECK PHOTOEYE
PE_10081   : FB_PhotoEye;  //S2140-01 TRIGGER PE & PINSTOP CLEAR PHOTOEYE
PE_10091   : FB_PhotoEye;  //P2140 EXIT PEPHOTOEYE
PE_10151   : FB_PhotoEye;  //P2140 JAM PEPHOTOEYE
PE_10291   : FB_PhotoEye;  //P2135 EXIT PEPHOTOEYE
PE_10302   : FB_PhotoEye;  //S2141-01 TRIGGER PHOTOEYE
PE_11191   : FB_PhotoEye;  //P2140 SINGULATION TOTE DETECT PHOTOEYE
PE_11221   : FB_PhotoEye;  //P2140 SINGULATION GRAB TRIGGER PHOTOEYE
PE_11241   : FB_PhotoEye;  //P2140 FULL PEPHOTOEYE
PE_12091   : FB_PhotoEye;  //P3085 EXIT PHOTOEYE
PE_12121   : FB_PhotoEye;  //P2130 FIRE DOOR PHOTOEYE
PE_12171   : FB_PhotoEye;  //P2130 DISCHARGE PHOTOEYE
PE_12181   : FB_PhotoEye;  //P3095 EXIT PHOTOEYE
PE_12271   : FB_PhotoEye;  //P3090 EXIT PHOTOEYE
END_VAR

 VAR PERSISTENT
	PE_10302OnTime: TIME := T#50MS;	
	PE_10081OnTime: TIME := T#50MS;
	PE_9161OnTime: TIME := T#135MS;
	PE_2301OnTime: TIME := T#175MS;
END_VAR

//P2150 FULL PHOTOEYE
PE_2101(
   In_Status:= ,
   CFG_PEOKState:= 1,
   CFG_OnDlyTime:= DebounceOnTime,
   CFG_OffDlyTime:= DebounceOffTime,
   CFG_JamDetTime:= JamDetectTime,
   In_Sim:=
);

//P2150 INDUCT PE SORTER PHOTOEYE
PE_2131(
   In_Status:= ,
   CFG_PEOKState:= 1,
   CFG_OnDlyTime:= DebounceOnTime,
   CFG_OffDlyTime:= DebounceOffTime,
   CFG_JamDetTime:= JamDetectTime,
   In_Sim:=
);

//P2146 FULL PHOTOEYE
PE_2201(
   In_Status:= Conveyors.P2146.Out_ConvCrntMtr,
   CFG_PEOKState:= 1,
   CFG_OnDlyTime:= DebounceOnTime,
   CFG_OffDlyTime:= DebounceOffTime,
   CFG_JamDetTime:= JamDetectTime,
   CFG_HoldWithStatus := TRUE,
   In_Sim:=
);

//P2145 EXIT PHOTOEYE
PE_2231(
   In_Status:= ,
   CFG_PEOKState:= 1,
   CFG_OnDlyTime:= DebounceOnTime,
   CFG_OffDlyTime:= DebounceOffTime,
   CFG_JamDetTime:= JamDetectTime,
   In_Sim:=
);

//S2150 TRIGGER PHOTOEYE
PE_2301(
   In_Status:= ,
   CFG_PEOKState:= 1,
   CFG_OnDlyTime:= PE_2301OnTime,
   CFG_OffDlyTime:= DebounceOffTime,
   CFG_JamDetTime:= JamDetectTime,
   In_Sim:=
);

//P2150 PE SINGULATION GRABBER TRIGGER PHOTOEYE
PE_2331(
   In_Status:= ,
   CFG_PEOKState:= 1,
   CFG_OnDlyTime:= DebounceOnTime,
   CFG_OffDlyTime:= DebounceOffTime,
   CFG_JamDetTime:= JamDetectTime,
   In_Sim:=
);

//P2150-02 TRANSFER COMPLETED PHOTOEYE
PE_3111(
   In_Status:= ,
   CFG_PEOKState:= 1,
   CFG_OnDlyTime:= DebounceOnTime,
   CFG_OffDlyTime:= DebounceOffTime,
   CFG_JamDetTime:= JamDetectTime,
   In_Sim:=
);

//P2150-01 TRANSFER COMPLETED PHOTOEYE
PE_3231(
   In_Status:= ,
   CFG_PEOKState:= 1,
   CFG_OnDlyTime:= DebounceOnTime,
   CFG_OffDlyTime:= DebounceOffTime,
   CFG_JamDetTime:= JamDetectTime,
   In_Sim:=
);

//P2150-04 TRANSFER COMPLETED PHOTOEYE
PE_4091(
   In_Status:= ,
   CFG_PEOKState:= 1,
   CFG_OnDlyTime:= DebounceOnTime,
   CFG_OffDlyTime:= DebounceOffTime,
   CFG_JamDetTime:= JamDetectTime,
   In_Sim:=
);

//P2150 SORTER DISCHARGE PHOTOEYE
PE_4161(
   In_Status:= ,
   CFG_PEOKState:= 1,
   CFG_OnDlyTime:= DebounceOnTime,
   CFG_OffDlyTime:= DebounceOffTime,
   CFG_JamDetTime:= JamDetectTime,
   In_Sim:=
);

//P2150-03 TRANSFER COMPLETED PHOTOEYE
PE_4201(
   In_Status:= ,
   CFG_PEOKState:= 1,
   CFG_OnDlyTime:= DebounceOnTime,
   CFG_OffDlyTime:= DebounceOffTime,
   CFG_JamDetTime:= JamDetectTime,
   In_Sim:=
);

//P2141 EXIT PHOTOEYE
PE_8131(
   In_Status:= Conveyors.P2141.Out_ConvCrntMtr,
   CFG_PEOKState:= 1,
   CFG_OnDlyTime:= DebounceOnTime,
   CFG_OffDlyTime:= DebounceOffTime,
   CFG_JamDetTime:= JamDetectTime,
   CFG_HoldWithStatus := TRUE,
   In_Sim:=
);

//P2142 FULL PHOTOEYE
PE_8141(
   In_Status:= ,
   CFG_PEOKState:= 1,
   CFG_OnDlyTime:= T#3S,
   CFG_OffDlyTime:= DebounceOffTime,
   CFG_JamDetTime:= JamDetectTime,
   In_Sim:=
);

//P2143 EXIT PHOTOEYE
PE_8161(
   In_Status:= Conveyors.P2143.Out_ConvCrntMtr,
   CFG_PEOKState:= 1,
   CFG_OnDlyTime:= DebounceOnTime,
   CFG_OffDlyTime:= DebounceOffTime,
   CFG_JamDetTime:= JamDetectTime,
   CFG_HoldWithStatus := TRUE,
   In_Sim:=
);

//P3080 EXIT PHOTOEYE
PE_9141(
   In_Status:= ,
   CFG_PEOKState:= 1,
   CFG_OnDlyTime:= DebounceOnTime,
   CFG_OffDlyTime:= DebounceOffTime,
   CFG_JamDetTime:= JamDetectTime,
   In_Sim:=
);

//S3080-01 TRIGGER PHOTOEYE
PE_9161(
   In_Status:= ,
   CFG_PEOKState:= 1,
   CFG_OnDlyTime:= PE_9161OnTime,
   CFG_OffDlyTime:= DebounceOffTime,
   CFG_JamDetTime:= JamDetectTime,
   In_Sim:=
);

//P3080 EXIT PHOTOEYE
PE_9191(
   In_Status:= Conveyors.P3080.Out_ConvCrntMtr,
   CFG_PEOKState:= 1,
   CFG_OnDlyTime:= DebounceOnTime,
   CFG_OffDlyTime:= DebounceOffTime,
   CFG_JamDetTime:= JamDetectTime,
   CFG_HoldWithStatus := TRUE,
   In_Sim:=
);

//P3080 HEIGHT CHECK PHOTOEYE
PE_9221(
   In_Status:= ,
   CFG_PEOKState:= 1,
   CFG_OnDlyTime:= DebounceOnTime,
   CFG_OffDlyTime:= DebounceOffTime,
   CFG_JamDetTime:= JamDetectTime,
   In_Sim:=
);

//S2140-01 TRIGGER PE & PINSTOP CLEAR PHOTOEYE
PE_10081(
   In_Status:= ,
   CFG_PEOKState:= 1,
   CFG_OnDlyTime:= PE_10081OnTime,
   CFG_OffDlyTime:= DebounceOffTime,
   CFG_JamDetTime:= JamDetectTime,
   In_Sim:=
);

//P2140 EXIT PEPHOTOEYE
PE_10091(
   In_Status:= ,
   CFG_PEOKState:= 1,
   CFG_OnDlyTime:= DebounceOnTime,
   CFG_OffDlyTime:= DebounceOffTime,
   CFG_JamDetTime:= JamDetectTime,
   In_Sim:=
);

//P2140 JAM PEPHOTOEYE
PE_10151(
   In_Status:= Conveyors.P2140_Status.Sts_IsRunning,
   CFG_PEOKState:= 1,
   CFG_OnDlyTime:= DebounceOnTime,
   CFG_OffDlyTime:= DebounceOffTime,
   CFG_JamDetTime:= T#10S,
   In_Sim:=
);

//P2135 EXIT PEPHOTOEYE
PE_10291(
   In_Status:= ,
   CFG_PEOKState:= 1,
   CFG_OnDlyTime:= DebounceOnTime,
   CFG_OffDlyTime:= DebounceOffTime,
   CFG_JamDetTime:= JamDetectTime,
   In_Sim:=
);

//S2141-01 TRIGGER PHOTOEYE
PE_10302(
   In_Status:= ,
   CFG_PEOKState:= 1,
   CFG_OnDlyTime:= PE_10302OnTime,
   CFG_OffDlyTime:= DebounceOffTime,
   CFG_JamDetTime:= JamDetectTime,
   In_Sim:=
);

//P2140 SINGULATION TOTE DETECT PHOTOEYE
PE_11191(
   In_Status:= ,
   CFG_PEOKState:= 1,
   CFG_OnDlyTime:= T#1000MS, // Delay the tote detection just shorter than the pin stop detection
   CFG_OffDlyTime:= DebounceOffTime,
   CFG_JamDetTime:= JamDetectTime,
   In_Sim:=
);

//P2140 SINGULATION GRAB TRIGGER PHOTOEYE
PE_11221(
   In_Status:= ,
   CFG_PEOKState:= 1,
   CFG_OnDlyTime:= T#1500MS,	// Use a custom delay at the pin stop
   CFG_OffDlyTime:= DebounceOffTime,
   CFG_JamDetTime:= JamDetectTime,
   In_Sim:=
);

//P2140 FULL PEP HOTOEYE
PE_11241(
   In_Status:= ,
   CFG_PEOKState:= 1,
   CFG_OnDlyTime:= DebounceOnTime,
   CFG_OffDlyTime:= DebounceOffTime,
   CFG_JamDetTime:= JamDetectTime,
   In_Sim:=
);

//P3085 EXIT PHOTOEYE
PE_12091(
   In_Status:= ,
   CFG_PEOKState:= 1,
   CFG_OnDlyTime:= DebounceOnTime,
   CFG_OffDlyTime:= DebounceOffTime,
   CFG_JamDetTime:= JamDetectTime,
   In_Sim:=
);

//P2130 FIRE DOOR PHOTOEYE
PE_12121(
   In_Status:= ,
   CFG_PEOKState:= 1,
   CFG_OnDlyTime:= DebounceOnTime,
   CFG_OffDlyTime:= DebounceOffTime,
   CFG_JamDetTime:= JamDetectTime,
   In_Sim:=
);

//P2130 DISCHARGE PHOTOEYE
PE_12171(
   In_Status:= ,
   CFG_PEOKState:= 1,
   CFG_OnDlyTime:= DebounceOnTime,
   CFG_OffDlyTime:= DebounceOffTime,
   CFG_JamDetTime:= JamDetectTime,
   In_Sim:=
);

//P3095 EXIT PHOTOEYE
PE_12181(
   In_Status:= ,
   CFG_PEOKState:= 1,
   CFG_OnDlyTime:= DebounceOnTime,
   CFG_OffDlyTime:= DebounceOffTime,
   CFG_JamDetTime:= JamDetectTime,
   In_Sim:=
);

//P3090 EXIT PHOTOEYE
PE_12271(
   In_Status:= ,
   CFG_PEOKState:= 1,
   CFG_OnDlyTime:= DebounceOnTime,
   CFG_OffDlyTime:= DebounceOffTime,
   CFG_JamDetTime:= JamDetectTime,
   In_Sim:=
);

END_PROGRAM

// ---- FunctionBlocks/Utils/FB_PhotoEye.TcPOU
FUNCTION_BLOCK FB_PhotoEye
(*
Function Block to combine the functionality of the Debounce Block and the 
	Jam Timer Block into one
*)
VAR_INPUT
	In_Status:	BOOL;		// Status to determine if Timer should run (like running status or State) (1=Watch for Jams)
	CFG_PEOKState: BOOL;		// The OK or ON State of the Input (0 or 1)
	CFG_OnDlyTime: TIME;		// Time to delay Output turning On after Input is On
	CFG_OffDlyTime: TIME;		// Time to delay Output turning Off after Input is Off
	CFG_JamDetTime: TIME;		// Time to wait before sending Jam detected Output
	CFG_HoldWithStatus: BOOL := FALSE;	// Hold Input state with Status input for items that are too samll to stop
	{attribute 'OPC.UA.DA' := '1'}
	In_Sim:	BOOL;		// Simulation Input Bit acts just like the input but can be forced from the program for testing
END_VAR
VAR_OUTPUT
	{attribute 'OPC.UA.DA' := '1'}
	Out:	BOOL;		// Output Based on ON or OK state
	{attribute 'OPC.UA.DA' := '1'}
	Out_OnFltrd:	BOOL;		// ON filtered Only Output
	{attribute 'OPC.UA.DA' := '1'}
	Out_OffFltrd:	BOOL;		// Off filtered Only OutPut
	Out_OnOffFltrd:	BOOL;		// Both On and Off Filtered Output 
	Sts_OnDlyActive:	BOOL;
	Sts_OffDlyActive:	BOOL;
	JamDetected:	BOOL;
END_VAR
VAR
	In_PE AT %I* : BOOL;		// Mapped IO input for PE
	{attribute 'OPC.UA.DA' := '0'}
	PEInFttr:	FB_DigDebnce;	
	{attribute 'OPC.UA.DA' := '0'}
	PEInJam: 	FB_JamDetect;
	InputHold_SR: SR;
	fStatusOff: F_TRIG;
	PE_State : BOOL;
END_VAR

// Get the PE_State such that a blocked PE is always ON
PE_State := (In_PE OR In_Sim) XOR CFG_PEOKState;

// Test for Input holding with Status for items that pass beyond the PE when the motor stops
IF CFG_HoldWithStatus THEN
	fStatusOff(CLK := In_Status);
	InputHold_SR(SET1 :=(fStatusOff.Q AND PE_State)
		, RESET := In_Status);
END_IF

// Filter the ON and OFF of a digital input
PEInFttr(
	In:= (PE_State OR InputHold_SR.Q1), 
	CFG_OKState:= 0, 
	CFG_OnDlyTime:= CFG_OnDlyTime, 
	CFG_OffDlyTime:= CFG_OffDlyTime, 
//	In_Sim:= In_Sim, 
	Out=> Out, 
	OutOnFltrd=> Out_OnFltrd, 
	OutOffFltrd=> Out_OffFltrd, 
	OutOnOffFltrd=> Out_OnOffFltrd, 
	Sts_OnDlyActive=> Sts_OnDlyActive, 
	Sts_OffDlyActive=> Sts_OffDlyActive);
	
	
// Watch the time the photo eye is blocked 
PEInJam(
//	In_PE:= (In_PE OR In_Sim), 
	In_PE:= (PE_State OR InputHold_SR.Q1), 
	In_Status:= In_Status, 
	CFG_PEOKState:= 0, 
	JamDetTime:= CFG_JamDetTime, 
	JamDetected=> JamDetected);

END_FUNCTION_BLOCK

// ---- FunctionBlocks/Utils/Filters/FB_DigDebnce.TcPOU
(*
Function Block to filter the ON and OFF of a digital input In
The normal OK state can be configured with CFG_OKState
The Times for the On and Off delays are configured by CFG_OnDlyTime and CFG_OffDlyTime
and can be simulated using the In_Sim input
If the input In goes true the output OutOnFltrd is set to true after the on delay time has elapsed
If the input In goes false the output CFG_OffDlyTime will be held on until the off delay time has elapsed
The output OutOnOffFltrd is delayed for both on and off as described above
The status outputs Sts_OnDlyActive and Sts_OffDlyActive show that the delays are active
*)
FUNCTION_BLOCK FB_DigDebnce
VAR_INPUT
	In:	BOOL;	// Digital Input
	CFG_OKState:	BOOL;		// The OK or ON State of the Input (0 or 1)
	CFG_OnDlyTime:	TIME;		// Time to delay Output turning On after Input is On
	CFG_OffDlyTime:	TIME;		// Time to delay Output turning Off after Input is Off
	In_Sim:	BOOL;		// Simulation Input Bit acts just like the input but can be forced from the program for testing
END_VAR
VAR_OUTPUT
	{attribute 'OPC.UA.DA' := '1'}
	Out:	BOOL;		// Output Based on ON or OK state
	OutOnFltrd:	BOOL;		// ON filtered Only Output
	OutOffFltrd:	BOOL;		// Off filtered Only OutPut
	OutOnOffFltrd:	BOOL;		// Both On and Off Filtered Output 
	Sts_OnDlyActive: BOOL;
	Sts_OffDlyActive: BOOL;
	Sts_OnOffDlyActive: BOOL;
END_VAR
VAR
	OnDly_Ton: TON;
	OffDlyTof: TOF;
	OnOffDlyTof: TOF;
	
END_VAR

// Compare to normal ON state
Out := (In OR In_Sim) XOR CFG_OKState;

// Setup On Delay
OnDly_Ton(IN:= Out, PT:= CFG_OnDlyTime , Q=> OutOnFltrd , ET=> );
Sts_OnDlyActive := Out <> OutOnFltrd;

//Setup Off Delay
OffDlyTof(IN:= Out , PT:= CFG_OffDlyTime , Q=> OutOffFltrd , ET=> );
Sts_OffDlyActive := Out <> OutOffFltrd;

//Setup Both On and Off Delayed
OnOffDlyTof(IN:= OutOnFltrd , PT:= CFG_OffDlyTime , Q=> OutOnOffFltrd , ET=> );
Sts_OnOffDlyActive := Out <> OutOnOffFltrd;

END_FUNCTION_BLOCK

// ---- FunctionBlocks/Utils/FB_JamDetect.TcPOU
FUNCTION_BLOCK FB_JamDetect
VAR_INPUT
	In_PE:	BOOL;		// Photo Eye Input
	In_Status:	BOOL;		// Status to determine if Timer should run (like running status or State) (1=Watch for Jams)
	CFG_PEOKState:	BOOL;		// Photo OK State ( State of Photo Eye for OK or Not blocked State State (1 or 0))
	JamDetTime: TIME;		// Time to wait before sending Jam detected Output
END_VAR
VAR_OUTPUT
	JamDetected:	BOOL;		// Out for Jam detected
END_VAR
VAR
	PhotoEyeBlocked: BOOL;
	JamTimer: TON;
	JamWatchEnable: BOOL;
	PE_ClearTrig: F_TRIG;
END_VAR

PhotoEyeBlocked := In_PE XOR CFG_PEOKState;
JamWatchEnable := In_Status AND PhotoEyeBlocked;

JamTimer(IN:= JamWatchEnable, PT:= JamDetTime , Q=>  , ET=> );

IF JamTimer.Q THEN
	JamDetected := TRUE;
END_IF

PE_ClearTrig(CLK:= PhotoEyeBlocked);

IF PE_ClearTrig.Q AND JamDetected THEN
	JamDetected := FALSE;
END_IF

END_FUNCTION_BLOCK

// ---- POUs/Conveyors.TcPOU
PROGRAM Conveyors
VAR
//This section sets the default values for the VFD
	DefaultVelocity: INT := 1800;
	DefaultVelocityThreshold: INT := 500;
	ResetAllDrives: BOOL;
	
//Conveyors Incoming 2000 (Purple line)
//Transport
//----------------------------------------P2130--------------------------------------------------------------
   cfgP2130Label:	STRING(20) :=  'P2130';
   cfgP2130SleepTime:	TIME := T#10M;
   cfgP2130JamDetectTime:	TIME := T#30S;
   P2130SleepWakeTrig: ARRAY[1..5] OF BOOL;
   P2130: FB_CnvyrCnfig_1;
   P2130_StatePB: ST_StateCntrlPB;
	{attribute 'OPC.UA.DA' := '0'}
   P2130_Status : ST_EquipmentStatus;
//Transport
//----------------------------------------P2135--------------------------------------------------------------
   cfgP2135Label:	STRING(20) :=  'P2135';
   cfgP2135SleepTime:	TIME := T#10M;
   cfgP2135JamDetectTime:	TIME := T#30S;
   P2135SleepWakeTrig: ARRAY[1..5] OF BOOL;
   P2135: FB_CnvyrCnfig_1;
   P2135_StatePB: ST_StateCntrlPB;
 	{attribute 'OPC.UA.DA' := '0'}
  P2135_Status : ST_EquipmentStatus;
//Transport
//----------------------------------------P2140--------------------------------------------------------------
   cfgP2140Label:	STRING(20) :=  'P2140';
   cfgP2140SleepTime:	TIME := T#10M;
   cfgP2140JamDetectTime:	TIME := T#30S;
   P2140SleepWakeTrig: ARRAY[1..5] OF BOOL;
   P2140: FB_CnvyrCnfig_1;
   P2140_StatePB: ST_StateCntrlPB;
	{attribute 'OPC.UA.DA' := '0'}
   P2140_Status : ST_EquipmentStatus;
//Transport
//----------------------------------------P2143--------------------------------------------------------------
   cfgP2143Label:	STRING(20) :=  'P2143';
   cfgP2143SleepTime:	TIME := T#10M;
   cfgP2143JamDetectTime:	TIME := T#30S;
   P2143SleepWakeTrig: ARRAY[1..5] OF BOOL;
   P2143: FB_CnvyrCnfig_1;
   P2143_StatePB: ST_StateCntrlPB;
	{attribute 'OPC.UA.DA' := '0'}
   P2143_Status : ST_EquipmentStatus;
//Spiral
//----------------------------------------P2141--------------------------------------------------------------
   cfgP2141Label:	STRING(20) :=  'P2141';
   cfgP2141SleepTime:	TIME := T#10M;
   cfgP2141JamDetectTime:	TIME := T#30S;
   P2141SleepWakeTrig: ARRAY[1..5] OF BOOL;
   P2141: FB_CnvyrCnfig_1;
   P2141_StatePB: ST_StateCntrlPB;
	{attribute 'OPC.UA.DA' := '0'}
   P2141_Status : ST_EquipmentStatus;
   P2141_VFD	:	VFD;
   Test_VFD_P2141: BOOL;
//Transport
//----------------------------------------P2142--------------------------------------------------------------
   cfgP2142Label:	STRING(20) :=  'P2142';
   cfgP2142SleepTime:	TIME := T#10M;
   cfgP2142JamDetectTime:	TIME := T#30S;
   P2142SleepWakeTrig: ARRAY[1..5] OF BOOL;
   P2142: FB_CnvyrCnfig_1;
   P2142_StatePB: ST_StateCntrlPB;
	{attribute 'OPC.UA.DA' := '0'}
   P2142_Status : ST_EquipmentStatus;
//Transport
//----------------------------------------P2145--------------------------------------------------------------
   cfgP2145Label:	STRING(20) :=  'P2145';
   cfgP2145SleepTime:	TIME := T#10M;
   cfgP2145JamDetectTime:	TIME := T#30S;
   P2145SleepWakeTrig: ARRAY[1..5] OF BOOL;
   P2145: FB_CnvyrCnfig_1;
   P2145_StatePB: ST_StateCntrlPB;
	{attribute 'OPC.UA.DA' := '0'}
  P2145_Status : ST_EquipmentStatus;
//Spiral
//----------------------------------------P2146--------------------------------------------------------------
   cfgP2146Label:	STRING(20) :=  'P2146';
   cfgP2146SleepTime:	TIME := T#10M;
   cfgP2146JamDetectTime:	TIME := T#30S;
   P2146SleepWakeTrig: ARRAY[1..5] OF BOOL;
   P2146: FB_CnvyrCnfig_1;
   P2146_StatePB: ST_StateCntrlPB;
	{attribute 'OPC.UA.DA' := '0'}
   P2146_Status : ST_EquipmentStatus;
   P2146_VFD	:	VFD;
   Test_VFD_P2146: BOOL;
//Sorter
//----------------------------------------P2150--------------------------------------------------------------
   cfgP2150Label:	STRING(20) :=  'P2150';
   cfgP2150SleepTime:	TIME := T#10M;
   cfgP2150JamDetectTime:	TIME := T#30S;
   P2150SleepWakeTrig: ARRAY[1..5] OF BOOL;
   P2150: FB_CnvyrCnfig_1;
   P2150_StatePB: ST_StateCntrlPB;
	{attribute 'OPC.UA.DA' := '0'}
   P2150_Status : ST_EquipmentStatus;
   
//Conveyors Incoming 3000 (Green line)
//Spiral
//----------------------------------------P3080--------------------------------------------------------------
   cfgP3080Label:	STRING(20) :=  'P3080';
   cfgP3080SleepTime:	TIME := T#10M;
   cfgP3080JamDetectTime:	TIME := T#30S;
   P3080SleepWakeTrig: ARRAY[1..5] OF BOOL;
   P3080: FB_CnvyrCnfig_1;
   P3080_StatePB: ST_StateCntrlPB;
	{attribute 'OPC.UA.DA' := '0'}
   P3080_Status : ST_EquipmentStatus;
   P3080_VFD	:	VFD;
   Test_VFD_P3080: BOOL;
   P3080_ResetWakeTmr : TON ; //Timer for holding the reset button to wake up Infeed Conveyor
//Transport
//----------------------------------------P3085--------------------------------------------------------------
   cfgP3085Label:	STRING(20) :=  'P3085';
   cfgP3085SleepTime:	TIME := T#10M;
   cfgP3085JamDetectTime:	TIME := T#30S;
   P3085SleepWakeTrig: ARRAY[1..5] OF BOOL;
   P3085: FB_CnvyrCnfig_1;
   P3085_StatePB: ST_StateCntrlPB;
	{attribute 'OPC.UA.DA' := '0'}
   P3085_Status : ST_EquipmentStatus;
//Transport
//----------------------------------------P3090--------------------------------------------------------------
   cfgP3090Label:	STRING(20) :=  'P3090';
   cfgP3090SleepTime:	TIME := T#10M;
   cfgP3090JamDetectTime:	TIME := T#30S;
   P3090SleepWakeTrig: ARRAY[1..5] OF BOOL;
   P3090: FB_CnvyrCnfig_1;
   P3090_StatePB: ST_StateCntrlPB;
	{attribute 'OPC.UA.DA' := '0'}
   P3090_Status : ST_EquipmentStatus;
//Transport
//----------------------------------------P3095--------------------------------------------------------------
   cfgP3095Label:	STRING(20) :=  'P3095';
   cfgP3095SleepTime:	TIME := T#10M;
   cfgP3095JamDetectTime:	TIME := T#30S;
   P3095SleepWakeTrig: ARRAY[1..5] OF BOOL;
   P3095: FB_CnvyrCnfig_1;
   P3095_StatePB: ST_StateCntrlPB;
	{attribute 'OPC.UA.DA' := '0'}
   P3095_Status : ST_EquipmentStatus;
   
 	ComStatus: INT;
END_VAR
 
